LIN {X 0,Y 499.912,Z 1008.402,A -85,B 0,C 180,E1 21822.944,E2 21822.944} C_VEL
LIN {X 0,Y 504.848,Z 990.59,A -85,B 0,C 180,E1 21821.614,E2 21821.614} C_VEL
LIN {X 0,Y 509.783,Z 971.635,A -85,B 0,C 180,E1 21820.361,E2 21820.361} C_VEL
LIN {X 0,Y 514.878,Z 950.68,A -85,B 0,C 180,E1 21819.156,E2 21819.156} C_VEL
LIN {X 0,Y 520.634,Z 924.438,A -85,B 0,C 180,E1 21817.879,E2 21817.879} C_VEL
LIN {X 0,Y 525.094,Z 900.885,A -85,B 0,C 180,E1 21816.94,E2 21816.94} C_VEL
LIN {X 0,Y 528.641,Z 879.529,A -85,B 0,C 180,E1 21816.234,E2 21816.234} C_VEL
LIN {X 0,Y 531.615,Z 858.391,A -85,B 0,C 180,E1 21815.659,E2 21815.659} C_VEL
LIN {X 0,Y 534.308,Z 834.905,A -85,B 0,C 180,E1 21815.156,E2 21815.156} C_VEL
LIN {X 0,Y 536.742,Z 798.959,A -85,B 0,C 180,E1 21814.559,E2 21814.559} C_VEL
LIN {X 0,Y 548.311,Z 577.211,A -85,B 0,C 180,E1 21811.168,E2 21811.168} C_VEL
LIN {X 0,Y 553.738,Z 476.421,A -85,B 0,C 180,E1 21809.595,E2 21809.595} C_VEL
LIN {X 0,Y 544.019,Z 460.747,A -85,B 0,C 180,E1 21807.325,E2 21807.325} C_VEL
LIN {X 0,Y 534.97,Z 447.007,A -85,B 0,C 180,E1 21804.987,E2 21804.987} C_VEL
LIN {X 0,Y 526.575,Z 434.757,A -85,B 0,C 180,E1 21802.555,E2 21802.555} C_VEL
LIN {X 0,Y 521.092,Z 427.175,A -85,B 0,C 180,E1 21800.793,E2 21800.793} C_VEL
LIN {X 0,Y 517.186,Z 421.826,A -85,B 0,C 180,E1 21799.423,E2 21799.423} C_VEL
LIN {X 0,Y 512.336,Z 415.199,A -85,B 0,C 180,E1 21797.549,E2 21797.549} C_VEL
LIN {X 0,Y 507.667,Z 409.451,A -85,B 0,C 180,E1 21795.537,E2 21795.537} C_VEL
LIN {X 0,Y 506.729,Z 408.307,A -85,B 0,C 180,E1 21795.098,E2 21795.098} C_VEL
LIN {X 0,Y 503.193,Z 404.431,A -85,B 0,C 180,E1 21793.327,E2 21793.327} C_VEL
LIN {X 0,Y 502.048,Z 402.516,A -85,B 0,C 180,E1 21792.655,E2 21792.655} C_VEL
LIN {X 0,Y 498.77,Z 399.704,A -85,B 0,C 180,E1 21790.687,E2 21790.687} C_VEL
LIN {X 0,Y 496.811,Z 396.193,A -85,B 0,C 180,E1 21789.149,E2 21789.149} C_VEL
LIN {X 0,Y 493.046,Z 393.345,A -85,B 0,C 180,E1 21785.586,E2 21785.586} C_VEL
LIN {X 0,Y 491.629,Z 389.721,A -85,B 0,C 180,E1 21782.798,E2 21782.798} C_VEL
LIN {X 0,Y 491.752,Z 389.93,A -85,B 0,C 180,E1 21776.386,E2 21776.386} C_VEL
LIN {X 0,Y 492.937,Z 393.135,A -85,B 0,C 180,E1 21774.062,E2 21774.062} C_VEL
LIN {X 0,Y 496.449,Z 396.076,A -85,B 0,C 180,E1 21770.611,E2 21770.611} C_VEL
LIN {X 0,Y 497.033,Z 396.632,A -85,B 0,C 180,E1 21770.154,E2 21770.154} C_VEL
LIN {X 0,Y 499.129,Z 400.183,A -85,B 0,C 180,E1 21768.561,E2 21768.561} C_VEL
LIN {X 0,Y 502.365,Z 403.011,A -85,B 0,C 180,E1 21766.651,E2 21766.651} C_VEL
LIN {X 0,Y 505.237,Z 407.088,A -85,B 0,C 180,E1 21765.091,E2 21765.091} C_VEL
LIN {X 0,Y 507.467,Z 409.19,A -85,B 0,C 180,E1 21764.049,E2 21764.049} C_VEL
LIN {X 0,Y 510.926,Z 413.582,A -85,B 0,C 180,E1 21762.518,E2 21762.518} C_VEL
LIN {X 0,Y 512.597,Z 415.426,A -85,B 0,C 180,E1 21761.843,E2 21761.843} C_VEL
LIN {X 0,Y 517.532,Z 421.592,A -85,B 0,C 180,E1 21759.973,E2 21759.973} C_VEL
LIN {X 0,Y 522.294,Z 427.58,A -85,B 0,C 180,E1 21758.346,E2 21758.346} C_VEL
LIN {X 0,Y 526.558,Z 433.053,A -85,B 0,C 180,E1 21757.002,E2 21757.002} C_VEL
LIN {X 0,Y 534.048,Z 442.795,A -85,B 0,C 180,E1 21754.849,E2 21754.849} C_VEL
LIN {X 0,Y 542.616,Z 454.591,A -85,B 0,C 180,E1 21752.628,E2 21752.628} C_VEL
LIN {X 0,Y 551.517,Z 467.214,A -85,B 0,C 180,E1 21750.543,E2 21750.543} C_VEL
LIN {X 0,Y 553.74,Z 470.858,A -85,B 0,C 180,E1 21750.04,E2 21750.04} C_VEL
LIN {X 0,Y 542.052,Z 685.81,A -85,B 0,C 180,E1 21746.741,E2 21746.741} C_VEL
LIN {X 0,Y 535.822,Z 802.377,A -85,B 0,C 180,E1 21744.945,E2 21744.945} C_VEL
LIN {X 0,Y 533.339,Z 829.272,A -85,B 0,C 180,E1 21744.423,E2 21744.423} C_VEL
LIN {X 0,Y 529.817,Z 855.856,A -85,B 0,C 180,E1 21743.712,E2 21743.712} C_VEL
LIN {X 0,Y 526.549,Z 876.447,A -85,B 0,C 180,E1 21743.03,E2 21743.03} C_VEL
LIN {X 0,Y 522.905,Z 896.374,A -85,B 0,C 180,E1 21742.247,E2 21742.247} C_VEL
LIN {X 0,Y 518.74,Z 916.594,A -85,B 0,C 180,E1 21741.318,E2 21741.318} C_VEL
LIN {X 0,Y 514.01,Z 937.364,A -85,B 0,C 180,E1 21740.207,E2 21740.207} C_VEL
LIN {X 0,Y 507.632,Z 962.474,A -85,B 0,C 180,E1 21738.628,E2 21738.628} C_VEL
LIN {X 0,Y 501.992,Z 982.688,A -85,B 0,C 180,E1 21737.136,E2 21737.136} C_VEL
LIN {X 0,Y 496.85,Z 1000.115,A -85,B 0,C 180,E1 21735.676,E2 21735.676} C_VEL
LIN {X 0,Y 491.606,Z 1017.106,A -85,B 0,C 180,E1 21734.073,E2 21734.073} C_VEL
LIN {X 0,Y 486.038,Z 1034.545,A -85,B 0,C 180,E1 21732.217,E2 21732.217} C_VEL
LIN {X 0,Y 479.163,Z 1055.51,A -85,B 0,C 180,E1 21729.645,E2 21729.645} C_VEL
LIN {X 0,Y 473.899,Z 1071.228,A -85,B 0,C 180,E1 21727.419,E2 21727.419} C_VEL
LIN {X 0,Y 469.143,Z 1085.554,A -85,B 0,C 180,E1 21725.13,E2 21725.13} C_VEL
LIN {X 0,Y 464.525,Z 1099.816,A -85,B 0,C 180,E1 21722.555,E2 21722.555} C_VEL
LIN {X 0,Y 459.689,Z 1115.448,A -85,B 0,C 180,E1 21719.28,E2 21719.28} C_VEL
LIN {X 0,Y 459.025,Z 1117.597,A -85,B 0,C 180,E1 21718.78,E2 21718.78} C_VEL
LIN {X 0,Y 457.031,Z 1121.397,A -85,B 0,C 180,E1 21717.965,E2 21717.965} C_VEL
LIN {X 0,Y 448.52,Z 1131.236,A -85,B 0,C 180,E1 21715.841,E2 21715.841} C_VEL
LIN {X 0,Y 447.037,Z 1133.995,A -85,B 0,C 180,E1 21715.09,E2 21715.09} C_VEL
LIN {X 0,Y 444.634,Z 1143.256,A -85,B 0,C 180,E1 21712.196,E2 21712.196} C_VEL
LIN {X 0,Y 442.943,Z 1150.695,A -85,B 0,C 180,E1 21709.517,E2 21709.517} C_VEL
LIN {X 0,Y 441.679,Z 1157.301,A -85,B 0,C 180,E1 21706.742,E2 21706.742} C_VEL
LIN {X 0,Y 440.829,Z 1163.009,A -85,B 0,C 180,E1 21703.881,E2 21703.881} C_VEL
LIN {X 0,Y 440.237,Z 1168.647,A -85,B 0,C 180,E1 21700.336,E2 21700.336} C_VEL
LIN {X 0,Y 439.997,Z 1172.254,A -85,B 0,C 180,E1 21697.049,E2 21697.049} C_VEL
LIN {X 0,Y 439.929,Z 1174.329,A -85,B 0,C 180,E1 21694.171,E2 21694.171} C_VEL
LIN {X 0,Y 439.916,Z 1175.306,A -85,B 0,C 180,E1 21691.563,E2 21691.563} C_VEL
LIN {X 0,Y 439.916,Z 1175.409,A -85,B 0,C 180,E1 21688.958,E2 21688.958} C_VEL
LIN {X 0,Y 439.928,Z 1174.573,A -85,B 0,C 180,E1 21686.221,E2 21686.221} C_VEL
LIN {X 0,Y 439.98,Z 1172.771,A -85,B 0,C 180,E1 21683.476,E2 21683.476} C_VEL
LIN {X 0,Y 440.122,Z 1169.989,A -85,B 0,C 180,E1 21680.718,E2 21680.718} C_VEL
LIN {X 0,Y 440.447,Z 1166.205,A -85,B 0,C 180,E1 21677.945,E2 21677.945} C_VEL
LIN {X 0,Y 441.103,Z 1160.992,A -85,B 0,C 180,E1 21674.942,E2 21674.942} C_VEL
LIN {X 0,Y 442.567,Z 1152.645,A -85,B 0,C 180,E1 21671.151,E2 21671.151} C_VEL
LIN {X 0,Y 444.295,Z 1144.699,A -85,B 0,C 180,E1 21668.203,E2 21668.203} C_VEL
LIN {X 0,Y 446.381,Z 1136.332,A -85,B 0,C 180,E1 21665.519,E2 21665.519} C_VEL
LIN {X 0,Y 449.046,Z 1126.79,A -85,B 0,C 180,E1 21662.841,E2 21662.841} C_VEL
LIN {X 0,Y 452.729,Z 1114.867,A -85,B 0,C 180,E1 21659.912,E2 21659.912} C_VEL
LIN {X 0,Y 457.6,Z 1099.827,A -85,B 0,C 180,E1 21656.74,E2 21656.74} C_VEL
LIN {X 0,Y 462.204,Z 1086.291,A -85,B 0,C 180,E1 21654.263,E2 21654.263} C_VEL
LIN {X 0,Y 466.858,Z 1072.835,A -85,B 0,C 180,E1 21652.073,E2 21652.073} C_VEL
LIN {X 0,Y 472.19,Z 1057.515,A -85,B 0,C 180,E1 21649.858,E2 21649.858} C_VEL
LIN {X 0,Y 478.997,Z 1037.801,A -85,B 0,C 180,E1 21647.362,E2 21647.362} C_VEL
LIN {X 0,Y 485.502,Z 1018.081,A -85,B 0,C 180,E1 21645.225,E2 21645.225} C_VEL
LIN {X 0,Y 490.925,Z 1001.155,A -85,B 0,C 180,E1 21643.611,E2 21643.611} C_VEL
LIN {X 0,Y 496.235,Z 983.798,A -85,B 0,C 180,E1 21642.143,E2 21642.143} C_VEL
LIN {X 0,Y 501.578,Z 965.263,A -85,B 0,C 180,E1 21640.756,E2 21640.756} C_VEL
LIN {X 0,Y 508.144,Z 940.734,A -85,B 0,C 180,E1 21639.172,E2 21639.172} C_VEL
LIN {X 0,Y 513.483,Z 918.099,A -85,B 0,C 180,E1 21637.944,E2 21637.944} C_VEL
LIN {X 0,Y 517.761,Z 898.046,A -85,B 0,C 180,E1 21637.012,E2 21637.012} C_VEL
LIN {X 0,Y 521.64,Z 877.583,A -85,B 0,C 180,E1 21636.201,E2 21636.201} C_VEL
LIN {X 0,Y 525.123,Z 856.307,A -85,B 0,C 180,E1 21635.492,E2 21635.492} C_VEL
LIN {X 0,Y 528.747,Z 829.724,A -85,B 0,C 180,E1 21634.781,E2 21634.781} C_VEL
LIN {X 0,Y 531.309,Z 802.773,A -85,B 0,C 180,E1 21634.256,E2 21634.256} C_VEL
LIN {X 0,Y 537.398,Z 692.803,A -85,B 0,C 180,E1 21632.554,E2 21632.554} C_VEL
LIN {X 0,Y 549.515,Z 477.081,A -85,B 0,C 180,E1 21629.234,E2 21629.234} C_VEL
LIN {X 0,Y 549.54,Z 475.04,A -85,B 0,C 180,E1 21629.185,E2 21629.185} C_VEL
LIN {X 0,Y 540.335,Z 461.8,A -85,B 0,C 180,E1 21626.99,E2 21626.99} C_VEL
LIN {X 0,Y 531.088,Z 448.868,A -85,B 0,C 180,E1 21624.528,E2 21624.528} C_VEL
LIN {X 0,Y 522.239,Z 437.289,A -85,B 0,C 180,E1 21621.863,E2 21621.863} C_VEL
LIN {X 0,Y 518.024,Z 431.951,A -85,B 0,C 180,E1 21620.449,E2 21620.449} C_VEL
LIN {X 0,Y 513.95,Z 426.774,A -85,B 0,C 180,E1 21618.96,E2 21618.96} C_VEL
LIN {X 0,Y 509.921,Z 421.7,A -85,B 0,C 180,E1 21617.341,E2 21617.341} C_VEL
LIN {X 0,Y 506.344,Z 417.431,A -85,B 0,C 180,E1 21615.755,E2 21615.755} C_VEL
LIN {X 0,Y 505.081,Z 415.892,A -85,B 0,C 180,E1 21615.148,E2 21615.148} C_VEL
LIN {X 0,Y 501.861,Z 412.22,A -85,B 0,C 180,E1 21613.48,E2 21613.48} C_VEL
LIN {X 0,Y 500.543,Z 410.201,A -85,B 0,C 180,E1 21612.694,E2 21612.694} C_VEL
LIN {X 0,Y 497.092,Z 406.889,A -85,B 0,C 180,E1 21610.489,E2 21610.489} C_VEL
LIN {X 0,Y 495.664,Z 404.104,A -85,B 0,C 180,E1 21609.287,E2 21609.287} C_VEL
LIN {X 0,Y 491.91,Z 401.065,A -85,B 0,C 180,E1 21605.482,E2 21605.482} C_VEL
LIN {X 0,Y 490.704,Z 397.658,A -85,B 0,C 180,E1 21602.686,E2 21602.686} C_VEL
LIN {X 0,Y 490.802,Z 397.82,A -85,B 0,C 180,E1 21597.431,E2 21597.431} C_VEL
LIN {X 0,Y 492.462,Z 401.837,A -85,B 0,C 180,E1 21594.173,E2 21594.173} C_VEL
LIN {X 0,Y 495.879,Z 404.384,A -85,B 0,C 180,E1 21590.951,E2 21590.951} C_VEL
LIN {X 0,Y 498.399,Z 408.5,A -85,B 0,C 180,E1 21589.013,E2 21589.013} C_VEL
LIN {X 0,Y 501.04,Z 410.717,A -85,B 0,C 180,E1 21587.436,E2 21587.436} C_VEL
LIN {X 0,Y 504.069,Z 414.911,A -85,B 0,C 180,E1 21585.761,E2 21585.761} C_VEL
LIN {X 0,Y 506.142,Z 417.001,A -85,B 0,C 180,E1 21584.767,E2 21584.767} C_VEL
LIN {X 0,Y 509.665,Z 421.495,A -85,B 0,C 180,E1 21583.179,E2 21583.179} C_VEL
LIN {X 0,Y 514.337,Z 427.727,A -85,B 0,C 180,E1 21581.291,E2 21581.291} C_VEL
LIN {X 0,Y 518.996,Z 434.232,A -85,B 0,C 180,E1 21579.591,E2 21579.591} C_VEL
LIN {X 0,Y 524.613,Z 442.115,A -85,B 0,C 180,E1 21577.74,E2 21577.74} C_VEL
LIN {X 0,Y 533.804,Z 455.667,A -85,B 0,C 180,E1 21575.04,E2 21575.04} C_VEL
LIN {X 0,Y 542.974,Z 470.067,A -85,B 0,C 180,E1 21572.648,E2 21572.648} C_VEL
LIN {X 0,Y 549.68,Z 481.2,A -85,B 0,C 180,E1 21571.044,E2 21571.044} C_VEL
LIN {X 0,Y 537.951,Z 691.52,A -85,B 0,C 180,E1 21567.801,E2 21567.801} C_VEL
LIN {X 0,Y 530.83,Z 822.089,A -85,B 0,C 180,E1 21565.783,E2 21565.783} C_VEL
LIN {X 0,Y 528.193,Z 849.404,A -85,B 0,C 180,E1 21565.265,E2 21565.265} C_VEL
LIN {X 0,Y 524.46,Z 875.969,A -85,B 0,C 180,E1 21564.582,E2 21564.582} C_VEL
LIN {X 0,Y 520.839,Z 897.573,A -85,B 0,C 180,E1 21563.888,E2 21563.888} C_VEL
LIN {X 0,Y 516.962,Z 917.84,A -85,B 0,C 180,E1 21563.106,E2 21563.106} C_VEL
LIN {X 0,Y 512.59,Z 938.224,A -85,B 0,C 180,E1 21562.185,E2 21562.185} C_VEL
LIN {X 0,Y 506.938,Z 962.266,A -85,B 0,C 180,E1 21560.906,E2 21560.906} C_VEL
LIN {X 0,Y 500.544,Z 986.296,A -85,B 0,C 180,E1 21559.382,E2 21559.382} C_VEL
LIN {X 0,Y 495.148,Z 1005.224,A -85,B 0,C 180,E1 21557.997,E2 21557.997} C_VEL
LIN {X 0,Y 489.611,Z 1023.657,A -85,B 0,C 180,E1 21556.466,E2 21556.466} C_VEL
LIN {X 0,Y 483.812,Z 1042.239,A -85,B 0,C 180,E1 21554.715,E2 21554.715} C_VEL
LIN {X 0,Y 476.711,Z 1064.314,A -85,B 0,C 180,E1 21552.32,E2 21552.32} C_VEL
LIN {X 0,Y 471.001,Z 1081.529,A -85,B 0,C 180,E1 21550.16,E2 21550.16} C_VEL
LIN {X 0,Y 465.97,Z 1096.733,A -85,B 0,C 180,E1 21548.012,E2 21548.012} C_VEL
LIN {X 0,Y 461.4,Z 1110.664,A -85,B 0,C 180,E1 21545.809,E2 21545.809} C_VEL
LIN {X 0,Y 456.812,Z 1124.995,A -85,B 0,C 180,E1 21543.265,E2 21543.265} C_VEL
LIN {X 0,Y 451.799,Z 1141.559,A -85,B 0,C 180,E1 21539.864,E2 21539.864} C_VEL
LIN {X 0,Y 448.598,Z 1152.843,A -85,B 0,C 180,E1 21537.188,E2 21537.188} C_VEL
LIN {X 0,Y 446.003,Z 1162.97,A -85,B 0,C 180,E1 21534.465,E2 21534.465} C_VEL
LIN {X 0,Y 444.025,Z 1171.642,A -85,B 0,C 180,E1 21531.811,E2 21531.811} C_VEL
LIN {X 0,Y 442.381,Z 1180.02,A -85,B 0,C 180,E1 21528.857,E2 21528.857} C_VEL
LIN {X 0,Y 441.026,Z 1188.768,A -85,B 0,C 180,E1 21525.113,E2 21525.113} C_VEL
LIN {X 0,Y 440.386,Z 1194.411,A -85,B 0,C 180,E1 21522.057,E2 21522.057} C_VEL
LIN {X 0,Y 440.099,Z 1198.284,A -85,B 0,C 180,E1 21519.414,E2 21519.414} C_VEL
LIN {X 0,Y 439.966,Z 1201.265,A -85,B 0,C 180,E1 21516.707,E2 21516.707} C_VEL
LIN {X 0,Y 439.922,Z 1203.156,A -85,B 0,C 180,E1 21514.171,E2 21514.171} C_VEL
LIN {X 0,Y 439.919,Z 1204.182,A -85,B 0,C 180,E1 21511.563,E2 21511.563} C_VEL
LIN {X 0,Y 439.918,Z 1204.275,A -85,B 0,C 180,E1 21508.958,E2 21508.958} C_VEL
LIN {X 0,Y 439.921,Z 1203.436,A -85,B 0,C 180,E1 21506.351,E2 21506.351} C_VEL
LIN {X 0,Y 439.956,Z 1201.661,A -85,B 0,C 180,E1 21503.737,E2 21503.737} C_VEL
LIN {X 0,Y 440.064,Z 1198.942,A -85,B 0,C 180,E1 21501.112,E2 21501.112} C_VEL
LIN {X 0,Y 440.302,Z 1195.262,A -85,B 0,C 180,E1 21498.473,E2 21498.473} C_VEL
LIN {X 0,Y 440.826,Z 1190.339,A -85,B 0,C 180,E1 21495.687,E2 21495.687} C_VEL
LIN {X 0,Y 441.601,Z 1184.614,A -85,B 0,C 180,E1 21493.018,E2 21493.018} C_VEL
LIN {X 0,Y 442.848,Z 1177.481,A -85,B 0,C 180,E1 21490.204,E2 21490.204} C_VEL
LIN {X 0,Y 444.98,Z 1167.492,A -85,B 0,C 180,E1 21486.845,E2 21486.845} C_VEL
LIN {X 0,Y 447.908,Z 1155.482,A -85,B 0,C 180,E1 21483.484,E2 21483.484} C_VEL
LIN {X 0,Y 450.918,Z 1144.49,A -85,B 0,C 180,E1 21480.802,E2 21480.802} C_VEL
LIN {X 0,Y 454.409,Z 1132.778,A -85,B 0,C 180,E1 21478.272,E2 21478.272} C_VEL
LIN {X 0,Y 458.714,Z 1118.999,A -85,B 0,C 180,E1 21475.63,E2 21475.63} C_VEL
LIN {X 0,Y 464.839,Z 1100.155,A -85,B 0,C 180,E1 21472.503,E2 21472.503} C_VEL
LIN {X 0,Y 469.959,Z 1084.615,A -85,B 0,C 180,E1 21470.259,E2 21470.259} C_VEL
LIN {X 0,Y 475.065,Z 1069.163,A -85,B 0,C 180,E1 21468.27,E2 21468.27} C_VEL
LIN {X 0,Y 480.327,Z 1053.064,A -85,B 0,C 180,E1 21466.422,E2 21466.422} C_VEL
LIN {X 0,Y 486.799,Z 1032.9,A -85,B 0,C 180,E1 21464.376,E2 21464.376} C_VEL
LIN {X 0,Y 493.628,Z 1010.39,A -85,B 0,C 180,E1 21462.417,E2 21462.417} C_VEL
LIN {X 0,Y 499.161,Z 991.133,A -85,B 0,C 180,E1 21460.961,E2 21460.961} C_VEL
LIN {X 0,Y 504.246,Z 972.268,A -85,B 0,C 180,E1 21459.704,E2 21459.704} C_VEL
LIN {X 0,Y 509.328,Z 952.048,A -85,B 0,C 180,E1 21458.529,E2 21458.529} C_VEL
LIN {X 0,Y 514.893,Z 927.87,A -85,B 0,C 180,E1 21457.326,E2 21457.326} C_VEL
LIN {X 0,Y 519.986,Z 902.097,A -85,B 0,C 180,E1 21456.278,E2 21456.278} C_VEL
LIN {X 0,Y 523.759,Z 880.125,A -85,B 0,C 180,E1 21455.546,E2 21455.546} C_VEL
LIN {X 0,Y 526.846,Z 858.886,A -85,B 0,C 180,E1 21454.965,E2 21454.965} C_VEL
LIN {X 0,Y 529.517,Z 836.418,A -85,B 0,C 180,E1 21454.479,E2 21454.479} C_VEL
LIN {X 0,Y 531.799,Z 806.687,A -85,B 0,C 180,E1 21453.968,E2 21453.968} C_VEL
LIN {X 0,Y 543.813,Z 583.563,A -85,B 0,C 180,E1 21450.544,E2 21450.544} C_VEL
LIN {X 0,Y 549.559,Z 480.937,A -85,B 0,C 180,E1 21448.945,E2 21448.945} C_VEL
LIN {X 0,Y 541.033,Z 467.045,A -85,B 0,C 180,E1 21446.893,E2 21446.893} C_VEL
LIN {X 0,Y 532.508,Z 453.893,A -85,B 0,C 180,E1 21444.636,E2 21444.636} C_VEL
LIN {X 0,Y 523.69,Z 440.758,A -85,B 0,C 180,E1 21442.006,E2 21442.006} C_VEL
LIN {X 0,Y 516.206,Z 430.294,A -85,B 0,C 180,E1 21439.461,E2 21439.461} C_VEL
LIN {X 0,Y 510.049,Z 421.85,A -85,B 0,C 180,E1 21437.042,E2 21437.042} C_VEL
LIN {X 0,Y 506.435,Z 417.562,A -85,B 0,C 180,E1 21435.459,E2 21435.459} C_VEL
LIN {X 0,Y 505.288,Z 416.012,A -85,B 0,C 180,E1 21434.907,E2 21434.907} C_VEL
LIN {X 0,Y 501.71,Z 411.973,A -85,B 0,C 180,E1 21433.074,E2 21433.074} C_VEL
LIN {X 0,Y 500.674,Z 410.284,A -85,B 0,C 180,E1 21432.456,E2 21432.456} C_VEL
LIN {X 0,Y 497.466,Z 407.395,A -85,B 0,C 180,E1 21430.481,E2 21430.481} C_VEL
LIN {X 0,Y 495.538,Z 404.029,A -85,B 0,C 180,E1 21428.938,E2 21428.938} C_VEL
LIN {X 0,Y 491.819,Z 400.953,A -85,B 0,C 180,E1 21425.249,E2 21425.249} C_VEL
LIN {X 0,Y 490.604,Z 397.655,A -85,B 0,C 180,E1 21422.687,E2 21422.687} C_VEL
LIN {X 0,Y 490.727,Z 397.822,A -85,B 0,C 180,E1 21416.495,E2 21416.495} C_VEL
LIN {X 0,Y 491.877,Z 401.014,A -85,B 0,C 180,E1 21414.166,E2 21414.166} C_VEL
LIN {X 0,Y 495.336,Z 403.967,A -85,B 0,C 180,E1 21410.707,E2 21410.707} C_VEL
LIN {X 0,Y 495.897,Z 404.652,A -85,B 0,C 180,E1 21410.249,E2 21410.249} C_VEL
LIN {X 0,Y 498.157,Z 408.263,A -85,B 0,C 180,E1 21408.538,E2 21408.538} C_VEL
LIN {X 0,Y 500.991,Z 410.741,A -85,B 0,C 180,E1 21406.849,E2 21406.849} C_VEL
LIN {X 0,Y 503.933,Z 414.892,A -85,B 0,C 180,E1 21405.228,E2 21405.228} C_VEL
LIN {X 0,Y 506.021,Z 416.947,A -85,B 0,C 180,E1 21404.235,E2 21404.235} C_VEL
LIN {X 0,Y 509.568,Z 421.394,A -85,B 0,C 180,E1 21402.647,E2 21402.647} C_VEL
LIN {X 0,Y 511.144,Z 423.284,A -85,B 0,C 180,E1 21401.996,E2 21401.996} C_VEL
LIN {X 0,Y 515.816,Z 429.165,A -85,B 0,C 180,E1 21400.199,E2 21400.199} C_VEL
LIN {X 0,Y 520.521,Z 435.161,A -85,B 0,C 180,E1 21398.564,E2 21398.564} C_VEL
LIN {X 0,Y 524.736,Z 440.655,A -85,B 0,C 180,E1 21397.214,E2 21397.214} C_VEL
LIN {X 0,Y 532.057,Z 450.329,A -85,B 0,C 180,E1 21395.075,E2 21395.075} C_VEL
LIN {X 0,Y 541.933,Z 464.002,A -85,B 0,C 180,E1 21392.502,E2 21392.502} C_VEL
LIN {X 0,Y 549.547,Z 475.251,A -85,B 0,C 180,E1 21390.7,E2 21390.7} C_VEL
LIN {X 0,Y 537.465,Z 690.469,A -85,B 0,C 180,E1 21387.387,E2 21387.387} C_VEL
LIN {X 0,Y 531.264,Z 802.665,A -85,B 0,C 180,E1 21385.652,E2 21385.652} C_VEL
LIN {X 0,Y 528.699,Z 829.702,A -85,B 0,C 180,E1 21385.126,E2 21385.126} C_VEL
LIN {X 0,Y 525.085,Z 856.24,A -85,B 0,C 180,E1 21384.416,E2 21384.416} C_VEL
LIN {X 0,Y 521.745,Z 876.722,A -85,B 0,C 180,E1 21383.737,E2 21383.737} C_VEL
LIN {X 0,Y 518,Z 896.649,A -85,B 0,C 180,E1 21382.954,E2 21382.954} C_VEL
LIN {X 0,Y 513.715,Z 916.867,A -85,B 0,C 180,E1 21382.023,E2 21382.023} C_VEL
LIN {X 0,Y 508.732,Z 938.119,A -85,B 0,C 180,E1 21380.882,E2 21380.882} C_VEL
LIN {X 0,Y 502.041,Z 963.551,A -85,B 0,C 180,E1 21379.27,E2 21379.27} C_VEL
LIN {X 0,Y 496.455,Z 982.963,A -85,B 0,C 180,E1 21377.829,E2 21377.829} C_VEL
LIN {X 0,Y 491.098,Z 1000.508,A -85,B 0,C 180,E1 21376.353,E2 21376.353} C_VEL
LIN {X 0,Y 485.677,Z 1017.467,A -85,B 0,C 180,E1 21374.743,E2 21374.743} C_VEL
LIN {X 0,Y 479.695,Z 1035.544,A -85,B 0,C 180,E1 21372.801,E2 21372.801} C_VEL
LIN {X 0,Y 472.544,Z 1056.483,A -85,B 0,C 180,E1 21370.192,E2 21370.192} C_VEL
LIN {X 0,Y 467.315,Z 1071.504,A -85,B 0,C 180,E1 21368.039,E2 21368.039} C_VEL
LIN {X 0,Y 462.621,Z 1085.073,A -85,B 0,C 180,E1 21365.853,E2 21365.853} C_VEL
LIN {X 0,Y 458.201,Z 1098.029,A -85,B 0,C 180,E1 21363.51,E2 21363.51} C_VEL
LIN {X 0,Y 453.76,Z 1111.547,A -85,B 0,C 180,E1 21360.744,E2 21360.744} C_VEL
LIN {X 0,Y 449.448,Z 1125.473,A -85,B 0,C 180,E1 21357.419,E2 21357.419} C_VEL
LIN {X 0,Y 447.037,Z 1133.995,A -85,B 0,C 180,E1 21355.09,E2 21355.09} C_VEL
LIN {X 0,Y 445.245,Z 1137.162,A -85,B 0,C 180,E1 21354.208,E2 21354.208} C_VEL
LIN {X 0,Y 437.242,Z 1145.592,A -85,B 0,C 180,E1 21351.896,E2 21351.896} C_VEL
LIN {X 0,Y 435.932,Z 1147.901,A -85,B 0,C 180,E1 21351.092,E2 21351.092} C_VEL
LIN {X 0,Y 434.05,Z 1156.467,A -85,B 0,C 180,E1 21347.564,E2 21347.564} C_VEL
LIN {X 0,Y 433.058,Z 1162.235,A -85,B 0,C 180,E1 21344.713,E2 21344.713} C_VEL
LIN {X 0,Y 432.444,Z 1166.938,A -85,B 0,C 180,E1 21341.875,E2 21341.875} C_VEL
LIN {X 0,Y 432.135,Z 1170.458,A -85,B 0,C 180,E1 21339.187,E2 21339.187} C_VEL
LIN {X 0,Y 431.99,Z 1173.068,A -85,B 0,C 180,E1 21336.512,E2 21336.512} C_VEL
LIN {X 0,Y 431.933,Z 1174.79,A -85,B 0,C 180,E1 21333.849,E2 21333.849} C_VEL
LIN {X 0,Y 431.922,Z 1175.634,A -85,B 0,C 180,E1 21331.194,E2 21331.194} C_VEL
LIN {X 0,Y 431.921,Z 1175.606,A -85,B 0,C 180,E1 21328.541,E2 21328.541} C_VEL
LIN {X 0,Y 431.936,Z 1174.704,A -85,B 0,C 180,E1 21325.885,E2 21325.885} C_VEL
LIN {X 0,Y 431.992,Z 1172.909,A -85,B 0,C 180,E1 21323.202,E2 21323.202} C_VEL
LIN {X 0,Y 432.161,Z 1170.099,A -85,B 0,C 180,E1 21320.411,E2 21320.411} C_VEL
LIN {X 0,Y 432.547,Z 1166.071,A -85,B 0,C 180,E1 21317.45,E2 21317.45} C_VEL
LIN {X 0,Y 433.503,Z 1159.61,A -85,B 0,C 180,E1 21313.795,E2 21313.795} C_VEL
LIN {X 0,Y 434.986,Z 1151.881,A -85,B 0,C 180,E1 21310.391,E2 21310.391} C_VEL
LIN {X 0,Y 436.807,Z 1144.178,A -85,B 0,C 180,E1 21307.526,E2 21307.526} C_VEL
LIN {X 0,Y 439.228,Z 1135.244,A -85,B 0,C 180,E1 21304.657,E2 21304.657} C_VEL
LIN {X 0,Y 442.983,Z 1122.999,A -85,B 0,C 180,E1 21301.265,E2 21301.265} C_VEL
LIN {X 0,Y 447.339,Z 1109.627,A -85,B 0,C 180,E1 21298.144,E2 21298.144} C_VEL
LIN {X 0,Y 451.619,Z 1097.346,A -85,B 0,C 180,E1 21295.629,E2 21295.629} C_VEL
LIN {X 0,Y 456.281,Z 1084.29,A -85,B 0,C 180,E1 21293.257,E2 21293.257} C_VEL
LIN {X 0,Y 462.532,Z 1067.138,A -85,B 0,C 180,E1 21290.512,E2 21290.512} C_VEL
LIN {X 0,Y 469.273,Z 1048.173,A -85,B 0,C 180,E1 21287.926,E2 21287.926} C_VEL
LIN {X 0,Y 474.953,Z 1032.044,A -85,B 0,C 180,E1 21285.996,E2 21285.996} C_VEL
LIN {X 0,Y 480.673,Z 1015.343,A -85,B 0,C 180,E1 21284.226,E2 21284.226} C_VEL
LIN {X 0,Y 487.439,Z 994.816,A -85,B 0,C 180,E1 21282.313,E2 21282.313} C_VEL
LIN {X 0,Y 494.524,Z 971.532,A -85,B 0,C 180,E1 21280.469,E2 21280.469} C_VEL
LIN {X 0,Y 500.073,Z 951.864,A -85,B 0,C 180,E1 21279.125,E2 21279.125} C_VEL
LIN {X 0,Y 505.263,Z 932.019,A -85,B 0,C 180,E1 21277.947,E2 21277.947} C_VEL
LIN {X 0,Y 510.079,Z 911.622,A -85,B 0,C 180,E1 21276.893,E2 21276.893} C_VEL
LIN {X 0,Y 515.728,Z 884.461,A -85,B 0,C 180,E1 21275.724,E2 21275.724} C_VEL
LIN {X 0,Y 519.774,Z 861.161,A -85,B 0,C 180,E1 21274.914,E2 21274.914} C_VEL
LIN {X 0,Y 522.895,Z 839.751,A -85,B 0,C 180,E1 21274.305,E2 21274.305} C_VEL
LIN {X 0,Y 525.433,Z 818.339,A -85,B 0,C 180,E1 21273.819,E2 21273.819} C_VEL
LIN {X 0,Y 527.636,Z 792.245,A -85,B 0,C 180,E1 21273.356,E2 21273.356} C_VEL
LIN {X 0,Y 540.214,Z 569.172,A -85,B 0,C 180,E1 21269.921,E2 21269.921} C_VEL
LIN {X 0,Y 545.457,Z 479.792,A -85,B 0,C 180,E1 21268.53,E2 21268.53} C_VEL
LIN {X 0,Y 535.139,Z 464.787,A -85,B 0,C 180,E1 21265.957,E2 21265.957} C_VEL
LIN {X 0,Y 527.262,Z 454.048,A -85,B 0,C 180,E1 21263.765,E2 21263.765} C_VEL
LIN {X 0,Y 520.299,Z 444.653,A -85,B 0,C 180,E1 21261.594,E2 21261.594} C_VEL
LIN {X 0,Y 515.994,Z 439.147,A -85,B 0,C 180,E1 21260.118,E2 21260.118} C_VEL
LIN {X 0,Y 512.274,Z 434.32,A -85,B 0,C 180,E1 21258.728,E2 21258.728} C_VEL
LIN {X 0,Y 508.171,Z 429.155,A -85,B 0,C 180,E1 21257.048,E2 21257.048} C_VEL
LIN {X 0,Y 504.567,Z 424.613,A -85,B 0,C 180,E1 21255.399,E2 21255.399} C_VEL
LIN {X 0,Y 500.298,Z 419.609,A -85,B 0,C 180,E1 21253.17,E2 21253.17} C_VEL
LIN {X 0,Y 499.384,Z 418.079,A -85,B 0,C 180,E1 21252.606,E2 21252.606} C_VEL
LIN {X 0,Y 495.958,Z 414.809,A -85,B 0,C 180,E1 21250.395,E2 21250.395} C_VEL
LIN {X 0,Y 494.403,Z 411.931,A -85,B 0,C 180,E1 21249.076,E2 21249.076} C_VEL
LIN {X 0,Y 490.781,Z 408.828,A -85,B 0,C 180,E1 21245.26,E2 21245.26} C_VEL
LIN {X 0,Y 489.689,Z 405.594,A -85,B 0,C 180,E1 21242.575,E2 21242.575} C_VEL
LIN {X 0,Y 489.786,Z 405.716,A -85,B 0,C 180,E1 21237.543,E2 21237.543} C_VEL
LIN {X 0,Y 491.486,Z 409.825,A -85,B 0,C 180,E1 21234.162,E2 21234.162} C_VEL
LIN {X 0,Y 494.688,Z 412.23,A -85,B 0,C 180,E1 21231.105,E2 21231.105} C_VEL
LIN {X 0,Y 497.255,Z 416.391,A -85,B 0,C 180,E1 21229.105,E2 21229.105} C_VEL
LIN {X 0,Y 499.764,Z 418.606,A -85,B 0,C 180,E1 21227.58,E2 21227.58} C_VEL
LIN {X 0,Y 502.99,Z 422.931,A -85,B 0,C 180,E1 21225.788,E2 21225.788} C_VEL
LIN {X 0,Y 504.695,Z 424.739,A -85,B 0,C 180,E1 21224.957,E2 21224.957} C_VEL
LIN {X 0,Y 508.31,Z 429.304,A -85,B 0,C 180,E1 21223.31,E2 21223.31} C_VEL
LIN {X 0,Y 512.926,Z 435.691,A -85,B 0,C 180,E1 21221.414,E2 21221.414} C_VEL
LIN {X 0,Y 519.084,Z 444.288,A -85,B 0,C 180,E1 21219.182,E2 21219.182} C_VEL
LIN {X 0,Y 526.497,Z 455.289,A -85,B 0,C 180,E1 21216.802,E2 21216.802} C_VEL
LIN {X 0,Y 534.421,Z 467.383,A -85,B 0,C 180,E1 21214.541,E2 21214.541} C_VEL
LIN {X 0,Y 543.827,Z 482.605,A -85,B 0,C 180,E1 21212.13,E2 21212.13} C_VEL
LIN {X 0,Y 545.542,Z 485.664,A -85,B 0,C 180,E1 21211.711,E2 21211.711} C_VEL
LIN {X 0,Y 533.343,Z 697.786,A -85,B 0,C 180,E1 21208.432,E2 21208.432} C_VEL
LIN {X 0,Y 526.337,Z 821.952,A -85,B 0,C 180,E1 21206.506,E2 21206.506} C_VEL
LIN {X 0,Y 523.605,Z 849.464,A -85,B 0,C 180,E1 21205.983,E2 21205.983} C_VEL
LIN {X 0,Y 519.767,Z 875.982,A -85,B 0,C 180,E1 21205.301,E2 21205.301} C_VEL
LIN {X 0,Y 516.195,Z 896.802,A -85,B 0,C 180,E1 21204.633,E2 21204.633} C_VEL
LIN {X 0,Y 512.136,Z 917.451,A -85,B 0,C 180,E1 21203.841,E2 21203.841} C_VEL
LIN {X 0,Y 507.616,Z 937.962,A -85,B 0,C 180,E1 21202.914,E2 21202.914} C_VEL
LIN {X 0,Y 501.789,Z 962.001,A -85,B 0,C 180,E1 21201.636,E2 21201.636} C_VEL
LIN {X 0,Y 495.192,Z 986.028,A -85,B 0,C 180,E1 21200.109,E2 21200.109} C_VEL
LIN {X 0,Y 489.62,Z 1004.955,A -85,B 0,C 180,E1 21198.72,E2 21198.72} C_VEL
LIN {X 0,Y 483.83,Z 1023.606,A -85,B 0,C 180,E1 21197.163,E2 21197.163} C_VEL
LIN {X 0,Y 477.714,Z 1042.521,A -85,B 0,C 180,E1 21195.367,E2 21195.367} C_VEL
LIN {X 0,Y 469.977,Z 1065.582,A -85,B 0,C 180,E1 21192.822,E2 21192.822} C_VEL
LIN {X 0,Y 464.243,Z 1082.224,A -85,B 0,C 180,E1 21190.699,E2 21190.699} C_VEL
LIN {X 0,Y 459.043,Z 1097.316,A -85,B 0,C 180,E1 21188.532,E2 21188.532} C_VEL
LIN {X 0,Y 454.044,Z 1111.956,A -85,B 0,C 180,E1 21186.169,E2 21186.169} C_VEL
LIN {X 0,Y 448.285,Z 1129.263,A -85,B 0,C 180,E1 21182.971,E2 21182.971} C_VEL
LIN {X 0,Y 444.131,Z 1142.453,A -85,B 0,C 180,E1 21180.134,E2 21180.134} C_VEL
LIN {X 0,Y 440.829,Z 1153.62,A -85,B 0,C 180,E1 21177.415,E2 21177.415} C_VEL
LIN {X 0,Y 438.182,Z 1163.51,A -85,B 0,C 180,E1 21174.682,E2 21174.682} C_VEL
LIN {X 0,Y 435.761,Z 1173.859,A -85,B 0,C 180,E1 21171.397,E2 21171.397} C_VEL
LIN {X 0,Y 433.931,Z 1183.098,A -85,B 0,C 180,E1 21167.846,E2 21167.846} C_VEL
LIN {X 0,Y 432.954,Z 1189.546,A -85,B 0,C 180,E1 21164.853,E2 21164.853} C_VEL
LIN {X 0,Y 432.398,Z 1194.357,A -85,B 0,C 180,E1 21162.147,E2 21162.147} C_VEL
LIN {X 0,Y 432.102,Z 1198.183,A -85,B 0,C 180,E1 21159.456,E2 21159.456} C_VEL
LIN {X 0,Y 431.968,Z 1201.054,A -85,B 0,C 180,E1 21156.771,E2 21156.771} C_VEL
LIN {X 0,Y 431.925,Z 1202.963,A -85,B 0,C 180,E1 21154.115,E2 21154.115} C_VEL
LIN {X 0,Y 431.923,Z 1203.943,A -85,B 0,C 180,E1 21151.459,E2 21151.459} C_VEL
LIN {X 0,Y 431.922,Z 1204.013,A -85,B 0,C 180,E1 21148.939,E2 21148.939} C_VEL
LIN {X 0,Y 431.923,Z 1203.173,A -85,B 0,C 180,E1 21146.284,E2 21146.284} C_VEL
LIN {X 0,Y 431.962,Z 1201.397,A -85,B 0,C 180,E1 21143.621,E2 21143.621} C_VEL
LIN {X 0,Y 432.074,Z 1198.676,A -85,B 0,C 180,E1 21140.946,E2 21140.946} C_VEL
LIN {X 0,Y 432.334,Z 1194.995,A -85,B 0,C 180,E1 21138.257,E2 21138.257} C_VEL
LIN {X 0,Y 432.855,Z 1190.331,A -85,B 0,C 180,E1 21135.554,E2 21135.554} C_VEL
LIN {X 0,Y 433.67,Z 1184.655,A -85,B 0,C 180,E1 21132.836,E2 21132.836} C_VEL
LIN {X 0,Y 434.969,Z 1177.572,A -85,B 0,C 180,E1 21129.971,E2 21129.971} C_VEL
LIN {X 0,Y 436.902,Z 1168.78,A -85,B 0,C 180,E1 21126.929,E2 21126.929} C_VEL
LIN {X 0,Y 440.254,Z 1155.731,A -85,B 0,C 180,E1 21123.131,E2 21123.131} C_VEL
LIN {X 0,Y 443.404,Z 1144.797,A -85,B 0,C 180,E1 21120.407,E2 21120.407} C_VEL
LIN {X 0,Y 447.036,Z 1133.147,A -85,B 0,C 180,E1 21117.838,E2 21117.838} C_VEL
LIN {X 0,Y 451.269,Z 1120.145,A -85,B 0,C 180,E1 21115.29,E2 21115.29} C_VEL
LIN {X 0,Y 457.055,Z 1103.21,A -85,B 0,C 180,E1 21112.368,E2 21112.368} C_VEL
LIN {X 0,Y 463.184,Z 1085.276,A -85,B 0,C 180,E1 21109.72,E2 21109.72} C_VEL
LIN {X 0,Y 468.48,Z 1069.87,A -85,B 0,C 180,E1 21107.707,E2 21107.707} C_VEL
LIN {X 0,Y 473.944,Z 1053.785,A -85,B 0,C 180,E1 21105.833,E2 21105.833} C_VEL
LIN {X 0,Y 479.737,Z 1036.316,A -85,B 0,C 180,E1 21104.025,E2 21104.025} C_VEL
LIN {X 0,Y 486.975,Z 1013.786,A -85,B 0,C 180,E1 21101.99,E2 21101.99} C_VEL
LIN {X 0,Y 493.541,Z 991.674,A -85,B 0,C 180,E1 21100.293,E2 21100.293} C_VEL
LIN {X 0,Y 498.776,Z 972.899,A -85,B 0,C 180,E1 21099.032,E2 21099.032} C_VEL
LIN {X 0,Y 503.746,Z 953.798,A -85,B 0,C 180,E1 21097.91,E2 21097.91} C_VEL
LIN {X 0,Y 508.388,Z 934.423,A -85,B 0,C 180,E1 21096.92,E2 21096.92} C_VEL
LIN {X 0,Y 512.905,Z 913.55,A -85,B 0,C 180,E1 21096.002,E2 21096.002} C_VEL
LIN {X 0,Y 518.02,Z 886.601,A -85,B 0,C 180,E1 21095.023,E2 21095.023} C_VEL
LIN {X 0,Y 521.878,Z 861.445,A -85,B 0,C 180,E1 21094.309,E2 21094.309} C_VEL
LIN {X 0,Y 524.633,Z 839.466,A -85,B 0,C 180,E1 21093.82,E2 21093.82} C_VEL
LIN {X 0,Y 526.66,Z 816.733,A -85,B 0,C 180,E1 21093.411,E2 21093.411} C_VEL
LIN {X 0,Y 538.89,Z 598.341,A -85,B 0,C 180,E1 21090.039,E2 21090.039} C_VEL
LIN {X 0,Y 545.459,Z 485.383,A -85,B 0,C 180,E1 21088.285,E2 21088.285} C_VEL
LIN {X 0,Y 537.031,Z 471.684,A -85,B 0,C 180,E1 21086.185,E2 21086.185} C_VEL
LIN {X 0,Y 529.71,Z 460.26,A -85,B 0,C 180,E1 21084.181,E2 21084.181} C_VEL
LIN {X 0,Y 521.559,Z 447.909,A -85,B 0,C 180,E1 21081.686,E2 21081.686} C_VEL
LIN {X 0,Y 514.202,Z 437.479,A -85,B 0,C 180,E1 21079.127,E2 21079.127} C_VEL
LIN {X 0,Y 508.421,Z 429.423,A -85,B 0,C 180,E1 21076.804,E2 21076.804} C_VEL
LIN {X 0,Y 504.759,Z 424.925,A -85,B 0,C 180,E1 21075.158,E2 21075.158} C_VEL
LIN {X 0,Y 503.62,Z 423.525,A -85,B 0,C 180,E1 21074.605,E2 21074.605} C_VEL
LIN {X 0,Y 500.143,Z 419.359,A -85,B 0,C 180,E1 21072.763,E2 21072.763} C_VEL
LIN {X 0,Y 499.271,Z 418.025,A -85,B 0,C 180,E1 21072.236,E2 21072.236} C_VEL
LIN {X 0,Y 496.091,Z 414.971,A -85,B 0,C 180,E1 21070.217,E2 21070.217} C_VEL
LIN {X 0,Y 494.422,Z 411.923,A -85,B 0,C 180,E1 21068.841,E2 21068.841} C_VEL
LIN {X 0,Y 490.761,Z 408.831,A -85,B 0,C 180,E1 21065.143,E2 21065.143} C_VEL
LIN {X 0,Y 489.58,Z 405.589,A -85,B 0,C 180,E1 21062.575,E2 21062.575} C_VEL
LIN {X 0,Y 489.704,Z 405.716,A -85,B 0,C 180,E1 21056.605,E2 21056.605} C_VEL
LIN {X 0,Y 490.818,Z 408.893,A -85,B 0,C 180,E1 21054.271,E2 21054.271} C_VEL
LIN {X 0,Y 494.223,Z 411.857,A -85,B 0,C 180,E1 21050.803,E2 21050.803} C_VEL
LIN {X 0,Y 494.829,Z 412.798,A -85,B 0,C 180,E1 21050.286,E2 21050.286} C_VEL
LIN {X 0,Y 497.186,Z 416.33,A -85,B 0,C 180,E1 21048.516,E2 21048.516} C_VEL
LIN {X 0,Y 499.714,Z 418.64,A -85,B 0,C 180,E1 21046.991,E2 21046.991} C_VEL
LIN {X 0,Y 502.855,Z 422.914,A -85,B 0,C 180,E1 21045.255,E2 21045.255} C_VEL
LIN {X 0,Y 504.574,Z 424.686,A -85,B 0,C 180,E1 21044.424,E2 21044.424} C_VEL
LIN {X 0,Y 508.345,Z 429.324,A -85,B 0,C 180,E1 21042.722,E2 21042.722} C_VEL
LIN {X 0,Y 514.039,Z 436.631,A -85,B 0,C 180,E1 21040.454,E2 21040.454} C_VEL
LIN {X 0,Y 518.833,Z 442.842,A -85,B 0,C 180,E1 21038.758,E2 21038.758} C_VEL
LIN {X 0,Y 525.11,Z 451.03,A -85,B 0,C 180,E1 21036.757,E2 21036.757} C_VEL
LIN {X 0,Y 534.009,Z 463.321,A -85,B 0,C 180,E1 21034.223,E2 21034.223} C_VEL
LIN {X 0,Y 542.617,Z 475.745,A -85,B 0,C 180,E1 21032.032,E2 21032.032} C_VEL
LIN {X 0,Y 545.4,Z 480.1,A -85,B 0,C 180,E1 21031.362,E2 21031.362} C_VEL
LIN {X 0,Y 532.935,Z 695.343,A -85,B 0,C 180,E1 21028.042,E2 21028.042} C_VEL
LIN {X 0,Y 526.781,Z 803.059,A -85,B 0,C 180,E1 21026.369,E2 21026.369} C_VEL
LIN {X 0,Y 524.123,Z 830.268,A -85,B 0,C 180,E1 21025.838,E2 21025.838} C_VEL
LIN {X 0,Y 520.434,Z 856.624,A -85,B 0,C 180,E1 21025.132,E2 21025.132} C_VEL
LIN {X 0,Y 516.888,Z 877.731,A -85,B 0,C 180,E1 21024.43,E2 21024.43} C_VEL
LIN {X 0,Y 512.914,Z 898.2,A -85,B 0,C 180,E1 21023.619,E2 21023.619} C_VEL
LIN {X 0,Y 508.266,Z 919.386,A -85,B 0,C 180,E1 21022.631,E2 21022.631} C_VEL
LIN {X 0,Y 501.78,Z 945.528,A -85,B 0,C 180,E1 21021.179,E2 21021.179} C_VEL
LIN {X 0,Y 496.036,Z 966.236,A -85,B 0,C 180,E1 21019.813,E2 21019.813} C_VEL
LIN {X 0,Y 490.539,Z 984.691,A -85,B 0,C 180,E1 21018.422,E2 21018.422} C_VEL
LIN {X 0,Y 485.089,Z 1001.92,A -85,B 0,C 180,E1 21016.953,E2 21016.953} C_VEL
LIN {X 0,Y 479.28,Z 1019.46,A -85,B 0,C 180,E1 21015.262,E2 21015.262} C_VEL
LIN {X 0,Y 472.208,Z 1040.096,A -85,B 0,C 180,E1 21012.985,E2 21012.985} C_VEL
LIN {X 0,Y 465.553,Z 1058.583,A -85,B 0,C 180,E1 21010.598,E2 21010.598} C_VEL
LIN {X 0,Y 460.481,Z 1072.612,A -85,B 0,C 180,E1 21008.548,E2 21008.548} C_VEL
LIN {X 0,Y 455.618,Z 1086.107,A -85,B 0,C 180,E1 21006.336,E2 21006.336} C_VEL
LIN {X 0,Y 451.032,Z 1098.994,A -85,B 0,C 180,E1 21003.962,E2 21003.962} C_VEL
LIN {X 0,Y 445.925,Z 1113.965,A -85,B 0,C 180,E1 21000.818,E2 21000.818} C_VEL
LIN {X 0,Y 441.749,Z 1126.754,A -85,B 0,C 180,E1 20997.645,E2 20997.645} C_VEL
LIN {X 0,Y 438.918,Z 1136.324,A -85,B 0,C 180,E1 20994.925,E2 20994.925} C_VEL
LIN {X 0,Y 436.583,Z 1145.11,A -85,B 0,C 180,E1 20992.061,E2 20992.061} C_VEL
LIN {X 0,Y 435.932,Z 1147.901,A -85,B 0,C 180,E1 20991.092,E2 20991.092} C_VEL
LIN {X 0,Y 434.333,Z 1150.493,A -85,B 0,C 180,E1 20990.149,E2 20990.149} C_VEL
LIN {X 0,Y 426.846,Z 1157.175,A -85,B 0,C 180,E1 20987.654,E2 20987.654} C_VEL
LIN {X 0,Y 425.765,Z 1159.058,A -85,B 0,C 180,E1 20986.807,E2 20986.807} C_VEL
LIN {X 0,Y 424.649,Z 1166.006,A -85,B 0,C 180,E1 20982.925,E2 20982.925} C_VEL
LIN {X 0,Y 424.206,Z 1170.174,A -85,B 0,C 180,E1 20979.847,E2 20979.847} C_VEL
LIN {X 0,Y 424.013,Z 1173.004,A -85,B 0,C 180,E1 20977.043,E2 20977.043} C_VEL
LIN {X 0,Y 423.942,Z 1174.856,A -85,B 0,C 180,E1 20974.328,E2 20974.328} C_VEL
LIN {X 0,Y 423.924,Z 1175.831,A -85,B 0,C 180,E1 20971.622,E2 20971.622} C_VEL
LIN {X 0,Y 423.924,Z 1175.934,A -85,B 0,C 180,E1 20968.919,E2 20968.919} C_VEL
LIN {X 0,Y 423.94,Z 1175.098,A -85,B 0,C 180,E1 20966.078,E2 20966.078} C_VEL
LIN {X 0,Y 423.998,Z 1173.407,A -85,B 0,C 180,E1 20963.365,E2 20963.365} C_VEL
LIN {X 0,Y 424.152,Z 1170.827,A -85,B 0,C 180,E1 20960.639,E2 20960.639} C_VEL
LIN {X 0,Y 424.502,Z 1167.231,A -85,B 0,C 180,E1 20957.827,E2 20957.827} C_VEL
LIN {X 0,Y 425.132,Z 1162.665,A -85,B 0,C 180,E1 20955.007,E2 20955.007} C_VEL
LIN {X 0,Y 426.183,Z 1156.929,A -85,B 0,C 180,E1 20952.101,E2 20952.101} C_VEL
LIN {X 0,Y 427.894,Z 1149.399,A -85,B 0,C 180,E1 20948.909,E2 20948.909} C_VEL
LIN {X 0,Y 430.793,Z 1138.666,A -85,B 0,C 180,E1 20945.159,E2 20945.159} C_VEL
LIN {X 0,Y 433.797,Z 1128.842,A -85,B 0,C 180,E1 20942.252,E2 20942.252} C_VEL
LIN {X 0,Y 437.358,Z 1118.217,A -85,B 0,C 180,E1 20939.501,E2 20939.501} C_VEL
LIN {X 0,Y 441.59,Z 1106.246,A -85,B 0,C 180,E1 20936.774,E2 20936.774} C_VEL
LIN {X 0,Y 447.935,Z 1089.104,A -85,B 0,C 180,E1 20933.417,E2 20933.417} C_VEL
LIN {X 0,Y 453.208,Z 1075.039,A -85,B 0,C 180,E1 20931.041,E2 20931.041} C_VEL
LIN {X 0,Y 458.752,Z 1060.298,A -85,B 0,C 180,E1 20928.836,E2 20928.836} C_VEL
LIN {X 0,Y 464.461,Z 1044.941,A -85,B 0,C 180,E1 20926.799,E2 20926.799} C_VEL
LIN {X 0,Y 471.49,Z 1025.735,A -85,B 0,C 180,E1 20924.559,E2 20924.559} C_VEL
LIN {X 0,Y 478.934,Z 1004.057,A -85,B 0,C 180,E1 20922.403,E2 20922.403} C_VEL
LIN {X 0,Y 484.69,Z 986.507,A -85,B 0,C 180,E1 20920.883,E2 20920.883} C_VEL
LIN {X 0,Y 490.143,Z 968.847,A -85,B 0,C 180,E1 20919.53,E2 20919.53} C_VEL
LIN {X 0,Y 495.722,Z 949.446,A -85,B 0,C 180,E1 20918.223,E2 20918.223} C_VEL
LIN {X 0,Y 502.132,Z 925.296,A -85,B 0,C 180,E1 20916.825,E2 20916.825} C_VEL
LIN {X 0,Y 507.932,Z 899.835,A -85,B 0,C 180,E1 20915.612,E2 20915.612} C_VEL
LIN {X 0,Y 512.015,Z 879.564,A -85,B 0,C 180,E1 20914.8,E2 20914.8} C_VEL
LIN {X 0,Y 515.65,Z 858.691,A -85,B 0,C 180,E1 20914.097,E2 20914.097} C_VEL
LIN {X 0,Y 518.882,Z 836.623,A -85,B 0,C 180,E1 20913.488,E2 20913.488} C_VEL
LIN {X 0,Y 522.008,Z 809.252,A -85,B 0,C 180,E1 20912.905,E2 20912.905} C_VEL
LIN {X 0,Y 524.925,Z 763.677,A -85,B 0,C 180,E1 20912.178,E2 20912.178} C_VEL
LIN {X 0,Y 537.946,Z 541.415,A -85,B 0,C 180,E1 20908.744,E2 20908.744} C_VEL
LIN {X 0,Y 541.395,Z 484.595,A -85,B 0,C 180,E1 20907.857,E2 20907.857} C_VEL
LIN {X 0,Y 532.463,Z 471.434,A -85,B 0,C 180,E1 20905.559,E2 20905.559} C_VEL
LIN {X 0,Y 524.983,Z 461.076,A -85,B 0,C 180,E1 20903.428,E2 20903.428} C_VEL
LIN {X 0,Y 518.212,Z 451.827,A -85,B 0,C 180,E1 20901.269,E2 20901.269} C_VEL
LIN {X 0,Y 513.982,Z 446.338,A -85,B 0,C 180,E1 20899.785,E2 20899.785} C_VEL
LIN {X 0,Y 510.33,Z 441.562,A -85,B 0,C 180,E1 20898.388,E2 20898.388} C_VEL
LIN {X 0,Y 506.691,Z 436.844,A -85,B 0,C 180,E1 20896.863,E2 20896.863} C_VEL
LIN {X 0,Y 503.023,Z 432.163,A -85,B 0,C 180,E1 20895.153,E2 20895.153} C_VEL
LIN {X 0,Y 498.932,Z 427.309,A -85,B 0,C 180,E1 20892.971,E2 20892.971} C_VEL
LIN {X 0,Y 497.834,Z 425.698,A -85,B 0,C 180,E1 20892.292,E2 20892.292} C_VEL
LIN {X 0,Y 494.534,Z 422.27,A -85,B 0,C 180,E1 20890.072,E2 20890.072} C_VEL
LIN {X 0,Y 493.15,Z 419.751,A -85,B 0,C 180,E1 20888.864,E2 20888.864} C_VEL
LIN {X 0,Y 489.591,Z 416.463,A -85,B 0,C 180,E1 20884.921,E2 20884.921} C_VEL
LIN {X 0,Y 488.675,Z 413.531,A -85,B 0,C 180,E1 20882.463,E2 20882.463} C_VEL
LIN {X 0,Y 488.795,Z 413.798,A -85,B 0,C 180,E1 20877.538,E2 20877.538} C_VEL
LIN {X 0,Y 490.8,Z 418.111,A -85,B 0,C 180,E1 20873.801,E2 20873.801} C_VEL
LIN {X 0,Y 493.562,Z 420.216,A -85,B 0,C 180,E1 20871.202,E2 20871.202} C_VEL
LIN {X 0,Y 496.282,Z 424.458,A -85,B 0,C 180,E1 20869.083,E2 20869.083} C_VEL
LIN {X 0,Y 498.406,Z 426.318,A -85,B 0,C 180,E1 20867.781,E2 20867.781} C_VEL
LIN {X 0,Y 501.689,Z 430.732,A -85,B 0,C 180,E1 20865.927,E2 20865.927} C_VEL
LIN {X 0,Y 503.255,Z 432.471,A -85,B 0,C 180,E1 20865.149,E2 20865.149} C_VEL
LIN {X 0,Y 508.343,Z 439.048,A -85,B 0,C 180,E1 20862.84,E2 20862.84} C_VEL
LIN {X 0,Y 514.412,Z 447.785,A -85,B 0,C 180,E1 20860.439,E2 20860.439} C_VEL
LIN {X 0,Y 520.269,Z 456.269,A -85,B 0,C 180,E1 20858.405,E2 20858.405} C_VEL
LIN {X 0,Y 529.163,Z 469.839,A -85,B 0,C 180,E1 20855.674,E2 20855.674} C_VEL
LIN {X 0,Y 538.388,Z 484.748,A -85,B 0,C 180,E1 20853.173,E2 20853.173} C_VEL
LIN {X 0,Y 541.467,Z 490.306,A -85,B 0,C 180,E1 20852.386,E2 20852.386} C_VEL
LIN {X 0,Y 528.873,Z 702.716,A -85,B 0,C 180,E1 20849.095,E2 20849.095} C_VEL
LIN {X 0,Y 521.937,Z 821.707,A -85,B 0,C 180,E1 20847.243,E2 20847.243} C_VEL
LIN {X 0,Y 519.139,Z 849.212,A -85,B 0,C 180,E1 20846.72,E2 20846.72} C_VEL
LIN {X 0,Y 515.193,Z 875.783,A -85,B 0,C 180,E1 20846.04,E2 20846.04} C_VEL
LIN {X 0,Y 511.407,Z 897.246,A -85,B 0,C 180,E1 20845.35,E2 20845.35} C_VEL
LIN {X 0,Y 507.253,Z 917.745,A -85,B 0,C 180,E1 20844.561,E2 20844.561} C_VEL
LIN {X 0,Y 502.486,Z 938.723,A -85,B 0,C 180,E1 20843.608,E2 20843.608} C_VEL
LIN {X 0,Y 496.214,Z 963.652,A -85,B 0,C 180,E1 20842.267,E2 20842.267} C_VEL
LIN {X 0,Y 489.681,Z 986.58,A -85,B 0,C 180,E1 20840.794,E2 20840.794} C_VEL
LIN {X 0,Y 483.917,Z 1005.519,A -85,B 0,C 180,E1 20839.393,E2 20839.393} C_VEL
LIN {X 0,Y 478.027,Z 1023.859,A -85,B 0,C 180,E1 20837.849,E2 20837.849} C_VEL
LIN {X 0,Y 471.225,Z 1044.2,A -85,B 0,C 180,E1 20835.894,E2 20835.894} C_VEL
LIN {X 0,Y 463.647,Z 1065.822,A -85,B 0,C 180,E1 20833.466,E2 20833.466} C_VEL
LIN {X 0,Y 457.781,Z 1082.204,A -85,B 0,C 180,E1 20831.353,E2 20831.353} C_VEL
LIN {X 0,Y 452.456,Z 1097.041,A -85,B 0,C 180,E1 20829.199,E2 20829.199} C_VEL
LIN {X 0,Y 447.239,Z 1111.68,A -85,B 0,C 180,E1 20826.809,E2 20826.809} C_VEL
LIN {X 0,Y 441.216,Z 1128.987,A -85,B 0,C 180,E1 20823.569,E2 20823.569} C_VEL
LIN {X 0,Y 436.699,Z 1142.644,A -85,B 0,C 180,E1 20820.58,E2 20820.58} C_VEL
LIN {X 0,Y 433.356,Z 1153.421,A -85,B 0,C 180,E1 20817.907,E2 20817.907} C_VEL
LIN {X 0,Y 430.508,Z 1163.506,A -85,B 0,C 180,E1 20815.067,E2 20815.067} C_VEL
LIN {X 0,Y 427.837,Z 1174.397,A -85,B 0,C 180,E1 20811.525,E2 20811.525} C_VEL
LIN {X 0,Y 426.007,Z 1183.138,A -85,B 0,C 180,E1 20808.048,E2 20808.048} C_VEL
LIN {X 0,Y 425.026,Z 1189.276,A -85,B 0,C 180,E1 20805.137,E2 20805.137} C_VEL
LIN {X 0,Y 424.431,Z 1194.089,A -85,B 0,C 180,E1 20802.379,E2 20802.379} C_VEL
LIN {X 0,Y 424.117,Z 1197.917,A -85,B 0,C 180,E1 20799.636,E2 20799.636} C_VEL
LIN {X 0,Y 423.973,Z 1200.782,A -85,B 0,C 180,E1 20796.908,E2 20796.908} C_VEL
LIN {X 0,Y 423.929,Z 1202.7,A -85,B 0,C 180,E1 20794.193,E2 20794.193} C_VEL
LIN {X 0,Y 423.927,Z 1203.68,A -85,B 0,C 180,E1 20791.487,E2 20791.487} C_VEL
LIN {X 0,Y 423.927,Z 1203.75,A -85,B 0,C 180,E1 20788.919,E2 20788.919} C_VEL
LIN {X 0,Y 423.927,Z 1202.91,A -85,B 0,C 180,E1 20786.213,E2 20786.213} C_VEL
LIN {X 0,Y 423.966,Z 1201.133,A -85,B 0,C 180,E1 20783.5,E2 20783.5} C_VEL
LIN {X 0,Y 424.086,Z 1198.411,A -85,B 0,C 180,E1 20780.774,E2 20780.774} C_VEL
LIN {X 0,Y 424.368,Z 1194.728,A -85,B 0,C 180,E1 20778.034,E2 20778.034} C_VEL
LIN {X 0,Y 424.953,Z 1189.8,A -85,B 0,C 180,E1 20775.14,E2 20775.14} C_VEL
LIN {X 0,Y 425.847,Z 1184.073,A -85,B 0,C 180,E1 20772.369,E2 20772.369} C_VEL
LIN {X 0,Y 427.276,Z 1176.81,A -85,B 0,C 180,E1 20769.401,E2 20769.401} C_VEL
LIN {X 0,Y 429.755,Z 1166.518,A -85,B 0,C 180,E1 20765.828,E2 20765.828} C_VEL
LIN {X 0,Y 432.917,Z 1154.923,A -85,B 0,C 180,E1 20762.488,E2 20762.488} C_VEL
LIN {X 0,Y 436.289,Z 1143.934,A -85,B 0,C 180,E1 20759.723,E2 20759.723} C_VEL
LIN {X 0,Y 440.102,Z 1132.22,A -85,B 0,C 180,E1 20757.114,E2 20757.114} C_VEL
LIN {X 0,Y 444.84,Z 1118.44,A -85,B 0,C 180,E1 20754.398,E2 20754.398} C_VEL
LIN {X 0,Y 451.552,Z 1099.596,A -85,B 0,C 180,E1 20751.198,E2 20751.198} C_VEL
LIN {X 0,Y 457.103,Z 1084.082,A -85,B 0,C 180,E1 20748.91,E2 20748.91} C_VEL
LIN {X 0,Y 462.546,Z 1068.871,A -85,B 0,C 180,E1 20746.916,E2 20746.916} C_VEL
LIN {X 0,Y 468.251,Z 1052.687,A -85,B 0,C 180,E1 20745.026,E2 20745.026} C_VEL
LIN {X 0,Y 474.828,Z 1033.576,A -85,B 0,C 180,E1 20743.056,E2 20743.056} C_VEL
LIN {X 0,Y 482.569,Z 1009.797,A -85,B 0,C 180,E1 20740.955,E2 20740.955} C_VEL
LIN {X 0,Y 488.468,Z 990.58,A -85,B 0,C 180,E1 20739.494,E2 20739.494} C_VEL
LIN {X 0,Y 493.761,Z 972.169,A -85,B 0,C 180,E1 20738.262,E2 20738.262} C_VEL
LIN {X 0,Y 499.005,Z 952.51,A -85,B 0,C 180,E1 20737.111,E2 20737.111} C_VEL
LIN {X 0,Y 504.057,Z 931.874,A -85,B 0,C 180,E1 20736.068,E2 20736.068} C_VEL
LIN {X 0,Y 509.901,Z 904.983,A -85,B 0,C 180,E1 20734.932,E2 20734.932} C_VEL
LIN {X 0,Y 514.336,Z 880.663,A -85,B 0,C 180,E1 20734.111,E2 20734.111} C_VEL
LIN {X 0,Y 517.662,Z 859.059,A -85,B 0,C 180,E1 20733.518,E2 20733.518} C_VEL
LIN {X 0,Y 520.44,Z 837.001,A -85,B 0,C 180,E1 20733.04,E2 20733.04} C_VEL
LIN {X 0,Y 522.775,Z 809.577,A -85,B 0,C 180,E1 20732.557,E2 20732.557} C_VEL
LIN {X 0,Y 535.621,Z 585.923,A -85,B 0,C 180,E1 20729.104,E2 20729.104} C_VEL
LIN {X 0,Y 541.318,Z 489.808,A -85,B 0,C 180,E1 20727.592,E2 20727.592} C_VEL
LIN {X 0,Y 532.02,Z 474.49,A -85,B 0,C 180,E1 20725.165,E2 20725.165} C_VEL
LIN {X 0,Y 524.134,Z 462.252,A -85,B 0,C 180,E1 20722.871,E2 20722.871} C_VEL
LIN {X 0,Y 516.441,Z 450.636,A -85,B 0,C 180,E1 20720.337,E2 20720.337} C_VEL
LIN {X 0,Y 509.24,Z 440.338,A -85,B 0,C 180,E1 20717.601,E2 20717.601} C_VEL
LIN {X 0,Y 506.159,Z 436.369,A -85,B 0,C 180,E1 20716.291,E2 20716.291} C_VEL
LIN {X 0,Y 502.195,Z 431.225,A -85,B 0,C 180,E1 20714.411,E2 20714.411} C_VEL
LIN {X 0,Y 498.682,Z 426.901,A -85,B 0,C 180,E1 20712.506,E2 20712.506} C_VEL
LIN {X 0,Y 497.748,Z 425.677,A -85,B 0,C 180,E1 20711.941,E2 20711.941} C_VEL
LIN {X 0,Y 494.653,Z 422.426,A -85,B 0,C 180,E1 20709.894,E2 20709.894} C_VEL
LIN {X 0,Y 493.159,Z 419.753,A -85,B 0,C 180,E1 20708.629,E2 20708.629} C_VEL
LIN {X 0,Y 489.631,Z 416.567,A -85,B 0,C 180,E1 20704.92,E2 20704.92} C_VEL
LIN {X 0,Y 488.559,Z 413.522,A -85,B 0,C 180,E1 20702.463,E2 20702.463} C_VEL
LIN {X 0,Y 488.682,Z 413.611,A -85,B 0,C 180,E1 20696.716,E2 20696.716} C_VEL
LIN {X 0,Y 489.841,Z 416.885,A -85,B 0,C 180,E1 20694.26,E2 20694.26} C_VEL
LIN {X 0,Y 493.448,Z 420.198,A -85,B 0,C 180,E1 20690.612,E2 20690.612} C_VEL
LIN {X 0,Y 495.703,Z 423.862,A -85,B 0,C 180,E1 20688.834,E2 20688.834} C_VEL
LIN {X 0,Y 498.352,Z 426.357,A -85,B 0,C 180,E1 20687.191,E2 20687.191} C_VEL
LIN {X 0,Y 501.555,Z 430.716,A -85,B 0,C 180,E1 20685.393,E2 20685.393} C_VEL
LIN {X 0,Y 503.134,Z 432.417,A -85,B 0,C 180,E1 20684.615,E2 20684.615} C_VEL
LIN {X 0,Y 506.992,Z 437.133,A -85,B 0,C 180,E1 20682.852,E2 20682.852} C_VEL
LIN {X 0,Y 512.481,Z 444.402,A -85,B 0,C 180,E1 20680.629,E2 20680.629} C_VEL
LIN {X 0,Y 517.152,Z 450.517,A -85,B 0,C 180,E1 20678.953,E2 20678.953} C_VEL
LIN {X 0,Y 523.109,Z 458.43,A -85,B 0,C 180,E1 20677.02,E2 20677.02} C_VEL
LIN {X 0,Y 531.718,Z 470.467,A -85,B 0,C 180,E1 20674.522,E2 20674.522} C_VEL
LIN {X 0,Y 540.217,Z 482.927,A -85,B 0,C 180,E1 20672.317,E2 20672.317} C_VEL
LIN {X 0,Y 541.333,Z 484.861,A -85,B 0,C 180,E1 20672.036,E2 20672.036} C_VEL
LIN {X 0,Y 528.408,Z 701.393,A -85,B 0,C 180,E1 20668.689,E2 20668.689} C_VEL
LIN {X 0,Y 522.382,Z 803.452,A -85,B 0,C 180,E1 20667.098,E2 20667.098} C_VEL
LIN {X 0,Y 519.628,Z 830.817,A -85,B 0,C 180,E1 20666.563,E2 20666.563} C_VEL
LIN {X 0,Y 515.884,Z 856.9,A -85,B 0,C 180,E1 20665.864,E2 20665.864} C_VEL
LIN {X 0,Y 512.246,Z 878.006,A -85,B 0,C 180,E1 20665.163,E2 20665.163} C_VEL
LIN {X 0,Y 508.167,Z 898.474,A -85,B 0,C 180,E1 20664.351,E2 20664.351} C_VEL
LIN {X 0,Y 503.132,Z 920.782,A -85,B 0,C 180,E1 20663.308,E2 20663.308} C_VEL
LIN {X 0,Y 496.209,Z 947.586,A -85,B 0,C 180,E1 20661.799,E2 20661.799} C_VEL
LIN {X 0,Y 490.59,Z 967.233,A -85,B 0,C 180,E1 20660.49,E2 20660.49} C_VEL
LIN {X 0,Y 485.137,Z 984.965,A -85,B 0,C 180,E1 20659.146,E2 20659.146} C_VEL
LIN {X 0,Y 479.434,Z 1002.417,A -85,B 0,C 180,E1 20657.651,E2 20657.651} C_VEL
LIN {X 0,Y 473.095,Z 1020.937,A -85,B 0,C 180,E1 20655.849,E2 20655.849} C_VEL
LIN {X 0,Y 465.224,Z 1042.87,A -85,B 0,C 180,E1 20653.367,E2 20653.367} C_VEL
LIN {X 0,Y 459.104,Z 1059.315,A -85,B 0,C 180,E1 20651.208,E2 20651.208} C_VEL
LIN {X 0,Y 453.684,Z 1073.72,A -85,B 0,C 180,E1 20649.072,E2 20649.072} C_VEL
LIN {X 0,Y 448.367,Z 1087.898,A -85,B 0,C 180,E1 20646.701,E2 20646.701} C_VEL
LIN {X 0,Y 442.43,Z 1104.006,A -85,B 0,C 180,E1 20643.62,E2 20643.62} C_VEL
LIN {X 0,Y 437.489,Z 1117.846,A -85,B 0,C 180,E1 20640.498,E2 20640.498} C_VEL
LIN {X 0,Y 433.926,Z 1128.447,A -85,B 0,C 180,E1 20637.767,E2 20637.767} C_VEL
LIN {X 0,Y 430.898,Z 1138.301,A -85,B 0,C 180,E1 20634.863,E2 20634.863} C_VEL
LIN {X 0,Y 428.051,Z 1148.834,A -85,B 0,C 180,E1 20631.226,E2 20631.226} C_VEL
LIN {X 0,Y 426.222,Z 1156.739,A -85,B 0,C 180,E1 20627.897,E2 20627.897} C_VEL
LIN {X 0,Y 425.765,Z 1159.058,A -85,B 0,C 180,E1 20626.807,E2 20626.807} C_VEL
LIN {X 0,Y 424.427,Z 1161.168,A -85,B 0,C 180,E1 20625.816,E2 20625.816} C_VEL
LIN {X 0,Y 417.342,Z 1166.362,A -85,B 0,C 180,E1 20623.092,E2 20623.092} C_VEL
LIN {X 0,Y 416.548,Z 1167.561,A -85,B 0,C 180,E1 20622.274,E2 20622.274} C_VEL
LIN {X 0,Y 416.165,Z 1171.299,A -85,B 0,C 180,E1 20619.263,E2 20619.263} C_VEL
LIN {X 0,Y 415.993,Z 1174.148,A -85,B 0,C 180,E1 20616.071,E2 20616.071} C_VEL
LIN {X 0,Y 415.932,Z 1175.965,A -85,B 0,C 180,E1 20612.48,E2 20612.48} C_VEL
LIN {X 0,Y 415.924,Z 1176.241,A -85,B 0,C 180,E1 20609.174,E2 20609.174} C_VEL
LIN {X 0,Y 415.943,Z 1175.493,A -85,B 0,C 180,E1 20606.279,E2 20606.279} C_VEL
LIN {X 0,Y 416.006,Z 1173.781,A -85,B 0,C 180,E1 20603.375,E2 20603.375} C_VEL
LIN {X 0,Y 416.179,Z 1171.092,A -85,B 0,C 180,E1 20600.458,E2 20600.458} C_VEL
LIN {X 0,Y 416.546,Z 1167.603,A -85,B 0,C 180,E1 20597.665,E2 20597.665} C_VEL
LIN {X 0,Y 417.197,Z 1163.179,A -85,B 0,C 180,E1 20594.857,E2 20594.857} C_VEL
LIN {X 0,Y 418.301,Z 1157.492,A -85,B 0,C 180,E1 20591.896,E2 20591.896} C_VEL
LIN {X 0,Y 419.909,Z 1150.7,A -85,B 0,C 180,E1 20588.928,E2 20588.928} C_VEL
LIN {X 0,Y 422.623,Z 1141.163,A -85,B 0,C 180,E1 20585.393,E2 20585.393} C_VEL
LIN {X 0,Y 426.274,Z 1129.617,A -85,B 0,C 180,E1 20581.871,E2 20581.871} C_VEL
LIN {X 0,Y 429.988,Z 1119.05,A -85,B 0,C 180,E1 20579.077,E2 20579.077} C_VEL
LIN {X 0,Y 434.147,Z 1107.762,A -85,B 0,C 180,E1 20576.446,E2 20576.446} C_VEL
LIN {X 0,Y 439.837,Z 1093.075,A -85,B 0,C 180,E1 20573.445,E2 20573.445} C_VEL
LIN {X 0,Y 446.439,Z 1076.141,A -85,B 0,C 180,E1 20570.502,E2 20570.502} C_VEL
LIN {X 0,Y 452.348,Z 1061.024,A -85,B 0,C 180,E1 20568.208,E2 20568.208} C_VEL
LIN {X 0,Y 458.066,Z 1046.21,A -85,B 0,C 180,E1 20566.216,E2 20566.216} C_VEL
LIN {X 0,Y 464.04,Z 1030.386,A -85,B 0,C 180,E1 20564.328,E2 20564.328} C_VEL
LIN {X 0,Y 471.564,Z 1009.857,A -85,B 0,C 180,E1 20562.18,E2 20562.18} C_VEL
LIN {X 0,Y 478.891,Z 988.226,A -85,B 0,C 180,E1 20560.261,E2 20560.261} C_VEL
LIN {X 0,Y 484.8,Z 969.711,A -85,B 0,C 180,E1 20558.829,E2 20558.829} C_VEL
LIN {X 0,Y 490.468,Z 950.6,A -85,B 0,C 180,E1 20557.533,E2 20557.533} C_VEL
LIN {X 0,Y 496.229,Z 929.546,A -85,B 0,C 180,E1 20556.297,E2 20556.297} C_VEL
LIN {X 0,Y 502.725,Z 902.644,A -85,B 0,C 180,E1 20554.974,E2 20554.974} C_VEL
LIN {X 0,Y 507.333,Z 880.48,A -85,B 0,C 180,E1 20554.078,E2 20554.078} C_VEL
LIN {X 0,Y 511.095,Z 859.505,A -85,B 0,C 180,E1 20553.368,E2 20553.368} C_VEL
LIN {X 0,Y 514.353,Z 837.911,A -85,B 0,C 180,E1 20552.769,E2 20552.769} C_VEL
LIN {X 0,Y 517.436,Z 812.256,A -85,B 0,C 180,E1 20552.211,E2 20552.211} C_VEL
LIN {X 0,Y 520.157,Z 773.303,A -85,B 0,C 180,E1 20551.578,E2 20551.578} C_VEL
LIN {X 0,Y 533.581,Z 550.612,A -85,B 0,C 180,E1 20548.13,E2 20548.13} C_VEL
LIN {X 0,Y 537.363,Z 489.299,A -85,B 0,C 180,E1 20547.161,E2 20547.161} C_VEL
LIN {X 0,Y 528.729,Z 476.521,A -85,B 0,C 180,E1 20544.854,E2 20544.854} C_VEL
LIN {X 0,Y 520.583,Z 464.989,A -85,B 0,C 180,E1 20542.412,E2 20542.412} C_VEL
LIN {X 0,Y 513.158,Z 454.925,A -85,B 0,C 180,E1 20539.878,E2 20539.878} C_VEL
LIN {X 0,Y 508.539,Z 448.952,A -85,B 0,C 180,E1 20538.099,E2 20538.099} C_VEL
LIN {X 0,Y 504.963,Z 444.291,A -85,B 0,C 180,E1 20536.567,E2 20536.567} C_VEL
LIN {X 0,Y 500.82,Z 439.006,A -85,B 0,C 180,E1 20534.57,E2 20534.57} C_VEL
LIN {X 0,Y 497.482,Z 434.854,A -85,B 0,C 180,E1 20532.714,E2 20532.714} C_VEL
LIN {X 0,Y 496.49,Z 433.44,A -85,B 0,C 180,E1 20532.09,E2 20532.09} C_VEL
LIN {X 0,Y 493.265,Z 429.961,A -85,B 0,C 180,E1 20529.863,E2 20529.863} C_VEL
LIN {X 0,Y 492.043,Z 427.64,A -85,B 0,C 180,E1 20528.767,E2 20528.767} C_VEL
LIN {X 0,Y 488.546,Z 424.341,A -85,B 0,C 180,E1 20524.814,E2 20524.814} C_VEL
LIN {X 0,Y 487.701,Z 421.471,A -85,B 0,C 180,E1 20522.468,E2 20522.468} C_VEL
LIN {X 0,Y 487.781,Z 421.688,A -85,B 0,C 180,E1 20517.65,E2 20517.65} C_VEL
LIN {X 0,Y 489.727,Z 425.992,A -85,B 0,C 180,E1 20513.905,E2 20513.905} C_VEL
LIN {X 0,Y 492.378,Z 428.049,A -85,B 0,C 180,E1 20511.357,E2 20511.357} C_VEL
LIN {X 0,Y 495.139,Z 432.344,A -85,B 0,C 180,E1 20509.175,E2 20509.175} C_VEL
LIN {X 0,Y 497.14,Z 434.19,A -85,B 0,C 180,E1 20507.926,E2 20507.926} C_VEL
LIN {X 0,Y 500.501,Z 438.638,A -85,B 0,C 180,E1 20506.011,E2 20506.011} C_VEL
LIN {X 0,Y 501.929,Z 440.377,A -85,B 0,C 180,E1 20505.286,E2 20505.286} C_VEL
LIN {X 0,Y 506.716,Z 446.595,A -85,B 0,C 180,E1 20503.079,E2 20503.079} C_VEL
LIN {X 0,Y 512.622,Z 455.255,A -85,B 0,C 180,E1 20500.694,E2 20500.694} C_VEL
LIN {X 0,Y 518.395,Z 463.778,A -85,B 0,C 180,E1 20498.65,E2 20498.65} C_VEL
LIN {X 0,Y 527.002,Z 477.148,A -85,B 0,C 180,E1 20495.955,E2 20495.955} C_VEL
LIN {X 0,Y 536.496,Z 492.704,A -85,B 0,C 180,E1 20493.34,E2 20493.34} C_VEL
LIN {X 0,Y 537.484,Z 494.703,A -85,B 0,C 180,E1 20493.075,E2 20493.075} C_VEL
LIN {X 0,Y 524.403,Z 708.85,A -85,B 0,C 180,E1 20489.751,E2 20489.751} C_VEL
LIN {X 0,Y 517.617,Z 821.569,A -85,B 0,C 180,E1 20487.991,E2 20487.991} C_VEL
LIN {X 0,Y 514.723,Z 849.235,A -85,B 0,C 180,E1 20487.464,E2 20487.464} C_VEL
LIN {X 0,Y 510.699,Z 875.636,A -85,B 0,C 180,E1 20486.789,E2 20486.789} C_VEL
LIN {X 0,Y 506.831,Z 897.03,A -85,B 0,C 180,E1 20486.103,E2 20486.103} C_VEL
LIN {X 0,Y 502.578,Z 917.456,A -85,B 0,C 180,E1 20485.319,E2 20485.319} C_VEL
LIN {X 0,Y 497.652,Z 938.568,A -85,B 0,C 180,E1 20484.361,E2 20484.361} C_VEL
LIN {X 0,Y 490.955,Z 964.294,A -85,B 0,C 180,E1 20482.971,E2 20482.971} C_VEL
LIN {X 0,Y 484.491,Z 986.313,A -85,B 0,C 180,E1 20481.553,E2 20481.553} C_VEL
LIN {X 0,Y 478.343,Z 1005.901,A -85,B 0,C 180,E1 20480.096,E2 20480.096} C_VEL
LIN {X 0,Y 472.271,Z 1024.196,A -85,B 0,C 180,E1 20478.544,E2 20478.544} C_VEL
LIN {X 0,Y 464.847,Z 1045.671,A -85,B 0,C 180,E1 20476.458,E2 20476.458} C_VEL
LIN {X 0,Y 457.189,Z 1066.575,A -85,B 0,C 180,E1 20474.063,E2 20474.063} C_VEL
LIN {X 0,Y 451.301,Z 1082.399,A -85,B 0,C 180,E1 20471.996,E2 20471.996} C_VEL
LIN {X 0,Y 445.615,Z 1097.624,A -85,B 0,C 180,E1 20469.753,E2 20469.753} C_VEL
LIN {X 0,Y 439.39,Z 1114.539,A -85,B 0,C 180,E1 20466.923,E2 20466.923} C_VEL
LIN {X 0,Y 433.481,Z 1130.653,A -85,B 0,C 180,E1 20463.772,E2 20463.772} C_VEL
LIN {X 0,Y 429.207,Z 1143.077,A -85,B 0,C 180,E1 20460.985,E2 20460.985} C_VEL
LIN {X 0,Y 425.633,Z 1154.122,A -85,B 0,C 180,E1 20458.175,E2 20458.175} C_VEL
LIN {X 0,Y 422.129,Z 1166.243,A -85,B 0,C 180,E1 20454.637,E2 20454.637} C_VEL
LIN {X 0,Y 419.555,Z 1176.303,A -85,B 0,C 180,E1 20451.091,E2 20451.091} C_VEL
LIN {X 0,Y 418.032,Z 1183.491,A -85,B 0,C 180,E1 20448.116,E2 20448.116} C_VEL
LIN {X 0,Y 417.027,Z 1189.531,A -85,B 0,C 180,E1 20445.149,E2 20445.149} C_VEL
LIN {X 0,Y 416.407,Z 1194.414,A -85,B 0,C 180,E1 20442.229,E2 20442.229} C_VEL
LIN {X 0,Y 416.088,Z 1198.311,A -85,B 0,C 180,E1 20439.265,E2 20439.265} C_VEL
LIN {X 0,Y 415.955,Z 1201.339,A -85,B 0,C 180,E1 20436.071,E2 20436.071} C_VEL
LIN {X 0,Y 415.929,Z 1203.251,A -85,B 0,C 180,E1 20432.48,E2 20432.48} C_VEL
LIN {X 0,Y 415.923,Z 1203.534,A -85,B 0,C 180,E1 20429.174,E2 20429.174} C_VEL
LIN {X 0,Y 415.93,Z 1202.717,A -85,B 0,C 180,E1 20426.279,E2 20426.279} C_VEL
LIN {X 0,Y 415.97,Z 1200.869,A -85,B 0,C 180,E1 20423.375,E2 20423.375} C_VEL
LIN {X 0,Y 416.099,Z 1198.145,A -85,B 0,C 180,E1 20420.596,E2 20420.596} C_VEL
LIN {X 0,Y 416.407,Z 1194.414,A -85,B 0,C 180,E1 20417.771,E2 20417.771} C_VEL
LIN {X 0,Y 417.027,Z 1189.531,A -85,B 0,C 180,E1 20414.851,E2 20414.851} C_VEL
LIN {X 0,Y 418.032,Z 1183.489,A -85,B 0,C 180,E1 20411.884,E2 20411.884} C_VEL
LIN {X 0,Y 419.557,Z 1176.3,A -85,B 0,C 180,E1 20408.909,E2 20408.909} C_VEL
LIN {X 0,Y 422.247,Z 1165.779,A -85,B 0,C 180,E1 20405.221,E2 20405.221} C_VEL
LIN {X 0,Y 425.635,Z 1154.124,A -85,B 0,C 180,E1 20401.825,E2 20401.825} C_VEL
LIN {X 0,Y 429.208,Z 1143.07,A -85,B 0,C 180,E1 20399.014,E2 20399.014} C_VEL
LIN {X 0,Y 433.479,Z 1130.645,A -85,B 0,C 180,E1 20396.228,E2 20396.228} C_VEL
LIN {X 0,Y 439.587,Z 1113.948,A -85,B 0,C 180,E1 20392.977,E2 20392.977} C_VEL
LIN {X 0,Y 445.611,Z 1097.598,A -85,B 0,C 180,E1 20390.247,E2 20390.247} C_VEL
LIN {X 0,Y 451.296,Z 1082.367,A -85,B 0,C 180,E1 20388.003,E2 20388.003} C_VEL
LIN {X 0,Y 457.374,Z 1066.022,A -85,B 0,C 180,E1 20385.872,E2 20385.872} C_VEL
LIN {X 0,Y 465.255,Z 1044.38,A -85,B 0,C 180,E1 20383.416,E2 20383.416} C_VEL
LIN {X 0,Y 472.261,Z 1024.119,A -85,B 0,C 180,E1 20381.455,E2 20381.455} C_VEL
LIN {X 0,Y 478.482,Z 1005.339,A -85,B 0,C 180,E1 20379.865,E2 20379.865} C_VEL
LIN {X 0,Y 484.77,Z 985.259,A -85,B 0,C 180,E1 20378.378,E2 20378.378} C_VEL
LIN {X 0,Y 491.985,Z 960.336,A -85,B 0,C 180,E1 20376.801,E2 20376.801} C_VEL
LIN {X 0,Y 497.909,Z 937.288,A -85,B 0,C 180,E1 20375.582,E2 20375.582} C_VEL
LIN {X 0,Y 502.698,Z 916.657,A -85,B 0,C 180,E1 20374.653,E2 20374.653} C_VEL
LIN {X 0,Y 506.964,Z 896.069,A -85,B 0,C 180,E1 20373.869,E2 20373.869} C_VEL
LIN {X 0,Y 510.982,Z 873.635,A -85,B 0,C 180,E1 20373.157,E2 20373.157} C_VEL
LIN {X 0,Y 515.197,Z 844.539,A -85,B 0,C 180,E1 20372.445,E2 20372.445} C_VEL
LIN {X 0,Y 517.646,Z 820.316,A -85,B 0,C 180,E1 20371.993,E2 20371.993} C_VEL
LIN {X 0,Y 530.056,Z 613.199,A -85,B 0,C 180,E1 20368.771,E2 20368.771} C_VEL
LIN {X 0,Y 537.376,Z 494.34,A -85,B 0,C 180,E1 20366.916,E2 20366.916} C_VEL
LIN {X 0,Y 527.596,Z 478.214,A -85,B 0,C 180,E1 20364.254,E2 20364.254} C_VEL
LIN {X 0,Y 519.221,Z 465.121,A -85,B 0,C 180,E1 20361.67,E2 20361.67} C_VEL
LIN {X 0,Y 513.062,Z 455.993,A -85,B 0,C 180,E1 20359.526,E2 20359.526} C_VEL
LIN {X 0,Y 507.334,Z 447.535,A -85,B 0,C 180,E1 20357.255,E2 20357.255} C_VEL
LIN {X 0,Y 504.437,Z 443.79,A -85,B 0,C 180,E1 20355.993,E2 20355.993} C_VEL
LIN {X 0,Y 500.776,Z 438.925,A -85,B 0,C 180,E1 20354.217,E2 20354.217} C_VEL
LIN {X 0,Y 497.231,Z 434.443,A -85,B 0,C 180,E1 20352.249,E2 20352.249} C_VEL
LIN {X 0,Y 496.399,Z 433.423,A -85,B 0,C 180,E1 20351.738,E2 20351.738} C_VEL
LIN {X 0,Y 493.303,Z 429.995,A -85,B 0,C 180,E1 20349.626,E2 20349.626} C_VEL
LIN {X 0,Y 492.047,Z 427.645,A -85,B 0,C 180,E1 20348.531,E2 20348.531} C_VEL
LIN {X 0,Y 488.577,Z 424.446,A -85,B 0,C 180,E1 20344.813,E2 20344.813} C_VEL
LIN {X 0,Y 487.585,Z 421.463,A -85,B 0,C 180,E1 20342.468,E2 20342.468} C_VEL
LIN {X 0,Y 487.663,Z 421.508,A -85,B 0,C 180,E1 20336.826,E2 20336.826} C_VEL
LIN {X 0,Y 488.784,Z 424.764,A -85,B 0,C 180,E1 20334.365,E2 20334.365} C_VEL
LIN {X 0,Y 492.262,Z 428.04,A -85,B 0,C 180,E1 20330.766,E2 20330.766} C_VEL
LIN {X 0,Y 494.731,Z 431.931,A -85,B 0,C 180,E1 20328.812,E2 20328.812} C_VEL
LIN {X 0,Y 497.084,Z 434.238,A -85,B 0,C 180,E1 20327.335,E2 20327.335} C_VEL
LIN {X 0,Y 500.368,Z 438.623,A -85,B 0,C 180,E1 20325.476,E2 20325.476} C_VEL
LIN {X 0,Y 501.808,Z 440.322,A -85,B 0,C 180,E1 20324.751,E2 20324.751} C_VEL
LIN {X 0,Y 506.374,Z 446.138,A -85,B 0,C 180,E1 20322.652,E2 20322.652} C_VEL
LIN {X 0,Y 510.791,Z 451.964,A -85,B 0,C 180,E1 20320.859,E2 20320.859} C_VEL
LIN {X 0,Y 517.271,Z 460.437,A -85,B 0,C 180,E1 20318.542,E2 20318.542} C_VEL
LIN {X 0,Y 527.565,Z 474.804,A -85,B 0,C 180,E1 20315.357,E2 20315.357} C_VEL
LIN {X 0,Y 537.151,Z 489.054,A -85,B 0,C 180,E1 20312.777,E2 20312.777} C_VEL
LIN {X 0,Y 537.326,Z 489.805,A -85,B 0,C 180,E1 20312.718,E2 20312.718} C_VEL
LIN {X 0,Y 524.036,Z 705.995,A -85,B 0,C 180,E1 20309.37,E2 20309.37} C_VEL
LIN {X 0,Y 518.077,Z 803.738,A -85,B 0,C 180,E1 20307.841,E2 20307.841} C_VEL
LIN {X 0,Y 515.255,Z 831.094,A -85,B 0,C 180,E1 20307.306,E2 20307.306} C_VEL
LIN {X 0,Y 511.42,Z 857.175,A -85,B 0,C 180,E1 20306.609,E2 20306.609} C_VEL
LIN {X 0,Y 507.688,Z 878.281,A -85,B 0,C 180,E1 20305.909,E2 20305.909} C_VEL
LIN {X 0,Y 503.506,Z 898.748,A -85,B 0,C 180,E1 20305.098,E2 20305.098} C_VEL
LIN {X 0,Y 498.599,Z 919.934,A -85,B 0,C 180,E1 20304.111,E2 20304.111} C_VEL
LIN {X 0,Y 491.752,Z 946.074,A -85,B 0,C 180,E1 20302.655,E2 20302.655} C_VEL
LIN {X 0,Y 485.664,Z 966.783,A -85,B 0,C 180,E1 20301.284,E2 20301.284} C_VEL
LIN {X 0,Y 480,Z 984.668,A -85,B 0,C 180,E1 20299.933,E2 20299.933} C_VEL
LIN {X 0,Y 474.202,Z 1001.876,A -85,B 0,C 180,E1 20298.462,E2 20298.462} C_VEL
LIN {X 0,Y 468.009,Z 1019.41,A -85,B 0,C 180,E1 20296.762,E2 20296.762} C_VEL
LIN {X 0,Y 460.605,Z 1039.63,A -85,B 0,C 180,E1 20294.519,E2 20294.519} C_VEL
LIN {X 0,Y 453.291,Z 1058.55,A -85,B 0,C 180,E1 20292.049,E2 20292.049} C_VEL
LIN {X 0,Y 447.572,Z 1073.166,A -85,B 0,C 180,E1 20289.877,E2 20289.877} C_VEL
LIN {X 0,Y 442.29,Z 1086.661,A -85,B 0,C 180,E1 20287.616,E2 20287.616} C_VEL
LIN {X 0,Y 436.928,Z 1100.528,A -85,B 0,C 180,E1 20284.988,E2 20284.988} C_VEL
LIN {X 0,Y 430.919,Z 1116.474,A -85,B 0,C 180,E1 20281.471,E2 20281.471} C_VEL
LIN {X 0,Y 426.892,Z 1127.808,A -85,B 0,C 180,E1 20278.542,E2 20278.542} C_VEL
LIN {X 0,Y 423.769,Z 1137.321,A -85,B 0,C 180,E1 20275.73,E2 20275.73} C_VEL
LIN {X 0,Y 421.066,Z 1146.447,A -85,B 0,C 180,E1 20272.624,E2 20272.624} C_VEL
LIN {X 0,Y 418.608,Z 1156.127,A -85,B 0,C 180,E1 20268.667,E2 20268.667} C_VEL
LIN {X 0,Y 417.317,Z 1162.528,A -85,B 0,C 180,E1 20265.423,E2 20265.423} C_VEL
LIN {X 0,Y 416.582,Z 1167.274,A -85,B 0,C 180,E1 20262.475,E2 20262.475} C_VEL
LIN {X 0,Y 416.548,Z 1167.561,A -85,B 0,C 180,E1 20262.274,E2 20262.274} C_VEL
LIN {X 0,Y 415.39,Z 1169.132,A -85,B 0,C 180,E1 20261.237,E2 20261.237} C_VEL
LIN {X 0,Y 408.624,Z 1172.744,A -85,B 0,C 180,E1 20258.308,E2 20258.308} C_VEL
LIN {X 0,Y 408.056,Z 1173.367,A -85,B 0,C 180,E1 20257.535,E2 20257.535} C_VEL
LIN {X 0,Y 407.954,Z 1175.384,A -85,B 0,C 180,E1 20254.498,E2 20254.498} C_VEL
LIN {X 0,Y 407.933,Z 1176.357,A -85,B 0,C 180,E1 20251.685,E2 20251.685} C_VEL
LIN {X 0,Y 407.933,Z 1176.459,A -85,B 0,C 180,E1 20248.876,E2 20248.876} C_VEL
LIN {X 0,Y 407.951,Z 1175.659,A -85,B 0,C 180,E1 20246.001,E2 20246.001} C_VEL
LIN {X 0,Y 408.019,Z 1173.934,A -85,B 0,C 180,E1 20243.104,E2 20243.104} C_VEL
LIN {X 0,Y 408.21,Z 1171.356,A -85,B 0,C 180,E1 20240.27,E2 20240.27} C_VEL
LIN {X 0,Y 408.631,Z 1167.669,A -85,B 0,C 180,E1 20237.278,E2 20237.278} C_VEL
LIN {X 0,Y 409.361,Z 1163.199,A -85,B 0,C 180,E1 20234.415,E2 20234.415} C_VEL
LIN {X 0,Y 410.602,Z 1157.299,A -85,B 0,C 180,E1 20231.314,E2 20231.314} C_VEL
LIN {X 0,Y 412.841,Z 1148.907,A -85,B 0,C 180,E1 20227.652,E2 20227.652} C_VEL
LIN {X 0,Y 415.932,Z 1138.713,A -85,B 0,C 180,E1 20224.039,E2 20224.039} C_VEL
LIN {X 0,Y 419.31,Z 1128.881,A -85,B 0,C 180,E1 20221.049,E2 20221.049} C_VEL
LIN {X 0,Y 423.262,Z 1118.2,A -85,B 0,C 180,E1 20218.212,E2 20218.212} C_VEL
LIN {X 0,Y 428.763,Z 1104.298,A -85,B 0,C 180,E1 20214.994,E2 20214.994} C_VEL
LIN {X 0,Y 434.948,Z 1088.889,A -85,B 0,C 180,E1 20211.97,E2 20211.97} C_VEL
LIN {X 0,Y 440.701,Z 1074.748,A -85,B 0,C 180,E1 20209.543,E2 20209.543} C_VEL
LIN {X 0,Y 446.731,Z 1059.925,A -85,B 0,C 180,E1 20207.3,E2 20207.3} C_VEL
LIN {X 0,Y 453.315,Z 1043.479,A -85,B 0,C 180,E1 20205.105,E2 20205.105} C_VEL
LIN {X 0,Y 461.755,Z 1021.551,A -85,B 0,C 180,E1 20202.59,E2 20202.59} C_VEL
LIN {X 0,Y 468.581,Z 1002.877,A -85,B 0,C 180,E1 20200.756,E2 20200.756} C_VEL
LIN {X 0,Y 474.845,Z 984.853,A -85,B 0,C 180,E1 20199.206,E2 20199.206} C_VEL
LIN {X 0,Y 480.894,Z 966.312,A -85,B 0,C 180,E1 20197.807,E2 20197.807} C_VEL
LIN {X 0,Y 487.995,Z 942.77,A -85,B 0,C 180,E1 20196.27,E2 20196.27} C_VEL
LIN {X 0,Y 494.214,Z 919.131,A -85,B 0,C 180,E1 20194.979,E2 20194.979} C_VEL
LIN {X 0,Y 498.984,Z 899.07,A -85,B 0,C 180,E1 20194.049,E2 20194.049} C_VEL
LIN {X 0,Y 503.279,Z 878.6,A -85,B 0,C 180,E1 20193.239,E2 20193.239} C_VEL
LIN {X 0,Y 507.203,Z 856.928,A -85,B 0,C 180,E1 20192.523,E2 20192.523} C_VEL
LIN {X 0,Y 511.202,Z 830.08,A -85,B 0,C 180,E1 20191.813,E2 20191.813} C_VEL
LIN {X 0,Y 513.968,Z 803.599,A -85,B 0,C 180,E1 20191.301,E2 20191.301} C_VEL
LIN {X 0,Y 521.778,Z 678.845,A -85,B 0,C 180,E1 20189.352,E2 20189.352} C_VEL
LIN {X 0,Y 533.502,Z 494.074,A -85,B 0,C 180,E1 20186.476,E2 20186.476} C_VEL
LIN {X 0,Y 524.121,Z 480.228,A -85,B 0,C 180,E1 20183.856,E2 20183.856} C_VEL
LIN {X 0,Y 515.169,Z 467.491,A -85,B 0,C 180,E1 20180.983,E2 20180.983} C_VEL
LIN {X 0,Y 507.57,Z 457.258,A -85,B 0,C 180,E1 20178.135,E2 20178.135} C_VEL
LIN {X 0,Y 503.249,Z 451.73,A -85,B 0,C 180,E1 20176.269,E2 20176.269} C_VEL
LIN {X 0,Y 499.411,Z 446.708,A -85,B 0,C 180,E1 20174.375,E2 20174.375} C_VEL
LIN {X 0,Y 496.042,Z 442.398,A -85,B 0,C 180,E1 20172.456,E2 20172.456} C_VEL
LIN {X 0,Y 495.152,Z 441.179,A -85,B 0,C 180,E1 20171.887,E2 20171.887} C_VEL
LIN {X 0,Y 492.003,Z 437.651,A -85,B 0,C 180,E1 20169.652,E2 20169.652} C_VEL
LIN {X 0,Y 490.801,Z 435.454,A -85,B 0,C 180,E1 20168.553,E2 20168.553} C_VEL
LIN {X 0,Y 487.441,Z 432.09,A -85,B 0,C 180,E1 20164.589,E2 20164.589} C_VEL
LIN {X 0,Y 486.689,Z 429.408,A -85,B 0,C 180,E1 20162.355,E2 20162.355} C_VEL
LIN {X 0,Y 486.77,Z 429.577,A -85,B 0,C 180,E1 20157.763,E2 20157.763} C_VEL
LIN {X 0,Y 488.753,Z 433.968,A -85,B 0,C 180,E1 20153.893,E2 20153.893} C_VEL
LIN {X 0,Y 491.199,Z 435.879,A -85,B 0,C 180,E1 20151.513,E2 20151.513} C_VEL
LIN {X 0,Y 493.997,Z 440.23,A -85,B 0,C 180,E1 20149.268,E2 20149.268} C_VEL
LIN {X 0,Y 495.878,Z 442.051,A -85,B 0,C 180,E1 20148.072,E2 20148.072} C_VEL
LIN {X 0,Y 499.315,Z 446.541,A -85,B 0,C 180,E1 20146.096,E2 20146.096} C_VEL
LIN {X 0,Y 500.93,Z 448.783,A -85,B 0,C 180,E1 20145.256,E2 20145.256} C_VEL
LIN {X 0,Y 505.098,Z 454.142,A -85,B 0,C 180,E1 20143.319,E2 20143.319} C_VEL
LIN {X 0,Y 510.913,Z 462.832,A -85,B 0,C 180,E1 20140.923,E2 20140.923} C_VEL
LIN {X 0,Y 516.763,Z 471.642,A -85,B 0,C 180,E1 20138.817,E2 20138.817} C_VEL
LIN {X 0,Y 524.94,Z 484.593,A -85,B 0,C 180,E1 20136.213,E2 20136.213} C_VEL
LIN {X 0,Y 533.583,Z 499.062,A -85,B 0,C 180,E1 20133.775,E2 20133.775} C_VEL
LIN {X 0,Y 520.037,Z 714.415,A -85,B 0,C 180,E1 20130.428,E2 20130.428} C_VEL
LIN {X 0,Y 513.386,Z 821.432,A -85,B 0,C 180,E1 20128.751,E2 20128.751} C_VEL
LIN {X 0,Y 510.414,Z 849.109,A -85,B 0,C 180,E1 20128.223,E2 20128.223} C_VEL
LIN {X 0,Y 506.315,Z 875.38,A -85,B 0,C 180,E1 20127.555,E2 20127.555} C_VEL
LIN {X 0,Y 502.353,Z 896.771,A -85,B 0,C 180,E1 20126.87,E2 20126.87} C_VEL
LIN {X 0,Y 498.049,Z 916.929,A -85,B 0,C 180,E1 20126.101,E2 20126.101} C_VEL
LIN {X 0,Y 493.211,Z 937.176,A -85,B 0,C 180,E1 20125.188,E2 20125.188} C_VEL
LIN {X 0,Y 486.826,Z 961.309,A -85,B 0,C 180,E1 20123.908,E2 20123.908} C_VEL
LIN {X 0,Y 479.65,Z 985.227,A -85,B 0,C 180,E1 20122.385,E2 20122.385} C_VEL
LIN {X 0,Y 473.308,Z 1004.891,A -85,B 0,C 180,E1 20120.926,E2 20120.926} C_VEL
LIN {X 0,Y 466.801,Z 1023.927,A -85,B 0,C 180,E1 20119.309,E2 20119.309} C_VEL
LIN {X 0,Y 459.009,Z 1045.707,A -85,B 0,C 180,E1 20117.183,E2 20117.183} C_VEL
LIN {X 0,Y 451.178,Z 1066.302,A -85,B 0,C 180,E1 20114.807,E2 20114.807} C_VEL
LIN {X 0,Y 445.057,Z 1082.138,A -85,B 0,C 180,E1 20112.721,E2 20112.721} C_VEL
LIN {X 0,Y 439.144,Z 1097.349,A -85,B 0,C 180,E1 20110.458,E2 20110.458} C_VEL
LIN {X 0,Y 432.542,Z 1114.573,A -85,B 0,C 180,E1 20107.542,E2 20107.542} C_VEL
LIN {X 0,Y 426.432,Z 1130.509,A -85,B 0,C 180,E1 20104.374,E2 20104.374} C_VEL
LIN {X 0,Y 421.979,Z 1142.796,A -85,B 0,C 180,E1 20101.577,E2 20101.577} C_VEL
LIN {X 0,Y 418.237,Z 1153.848,A -85,B 0,C 180,E1 20098.719,E2 20098.719} C_VEL
LIN {X 0,Y 414.526,Z 1165.969,A -85,B 0,C 180,E1 20095.12,E2 20095.12} C_VEL
LIN {X 0,Y 411.799,Z 1176.03,A -85,B 0,C 180,E1 20091.508,E2 20091.508} C_VEL
LIN {X 0,Y 410.177,Z 1183.22,A -85,B 0,C 180,E1 20088.475,E2 20088.475} C_VEL
LIN {X 0,Y 409.108,Z 1189.261,A -85,B 0,C 180,E1 20085.45,E2 20085.45} C_VEL
LIN {X 0,Y 408.458,Z 1193.98,A -85,B 0,C 180,E1 20082.583,E2 20082.583} C_VEL
LIN {X 0,Y 408.112,Z 1197.88,A -85,B 0,C 180,E1 20079.59,E2 20079.59} C_VEL
LIN {X 0,Y 407.971,Z 1200.723,A -85,B 0,C 180,E1 20076.614,E2 20076.614} C_VEL
LIN {X 0,Y 407.933,Z 1202.595,A -85,B 0,C 180,E1 20073.513,E2 20073.513} C_VEL
LIN {X 0,Y 407.937,Z 1203.403,A -85,B 0,C 180,E1 20070,E2 20070} C_VEL
LIN {X 0,Y 407.933,Z 1202.594,A -85,B 0,C 180,E1 20066.487,E2 20066.487} C_VEL
LIN {X 0,Y 407.971,Z 1200.722,A -85,B 0,C 180,E1 20063.386,E2 20063.386} C_VEL
LIN {X 0,Y 408.112,Z 1197.88,A -85,B 0,C 180,E1 20060.41,E2 20060.41} C_VEL
LIN {X 0,Y 408.458,Z 1193.98,A -85,B 0,C 180,E1 20057.417,E2 20057.417} C_VEL
LIN {X 0,Y 409.108,Z 1189.261,A -85,B 0,C 180,E1 20054.55,E2 20054.55} C_VEL
LIN {X 0,Y 410.177,Z 1183.217,A -85,B 0,C 180,E1 20051.525,E2 20051.525} C_VEL
LIN {X 0,Y 411.892,Z 1175.663,A -85,B 0,C 180,E1 20048.348,E2 20048.348} C_VEL
LIN {X 0,Y 414.912,Z 1164.564,A -85,B 0,C 180,E1 20044.447,E2 20044.447} C_VEL
LIN {X 0,Y 418.239,Z 1153.847,A -85,B 0,C 180,E1 20041.281,E2 20041.281} C_VEL
LIN {X 0,Y 421.979,Z 1142.791,A -85,B 0,C 180,E1 20038.423,E2 20038.423} C_VEL
LIN {X 0,Y 426.429,Z 1130.5,A -85,B 0,C 180,E1 20035.626,E2 20035.626} C_VEL
LIN {X 0,Y 432.648,Z 1114.24,A -85,B 0,C 180,E1 20032.403,E2 20032.403} C_VEL
LIN {X 0,Y 439.139,Z 1097.318,A -85,B 0,C 180,E1 20029.541,E2 20029.541} C_VEL
LIN {X 0,Y 445.056,Z 1082.087,A -85,B 0,C 180,E1 20027.276,E2 20027.276} C_VEL
LIN {X 0,Y 451.285,Z 1065.957,A -85,B 0,C 180,E1 20025.155,E2 20025.155} C_VEL
LIN {X 0,Y 459.327,Z 1044.718,A -85,B 0,C 180,E1 20022.721,E2 20022.721} C_VEL
LIN {X 0,Y 466.79,Z 1023.842,A -85,B 0,C 180,E1 20020.689,E2 20020.689} C_VEL
LIN {X 0,Y 473.296,Z 1004.79,A -85,B 0,C 180,E1 20019.072,E2 20019.072} C_VEL
LIN {X 0,Y 479.897,Z 984.297,A -85,B 0,C 180,E1 20017.556,E2 20017.556} C_VEL
LIN {X 0,Y 487.702,Z 957.791,A -85,B 0,C 180,E1 20015.899,E2 20015.899} C_VEL
LIN {X 0,Y 493.195,Z 937.013,A -85,B 0,C 180,E1 20014.809,E2 20014.809} C_VEL
LIN {X 0,Y 498.141,Z 916.256,A -85,B 0,C 180,E1 20013.877,E2 20013.877} C_VEL
LIN {X 0,Y 502.487,Z 895.794,A -85,B 0,C 180,E1 20013.101,E2 20013.101} C_VEL
LIN {X 0,Y 506.606,Z 873.36,A -85,B 0,C 180,E1 20012.392,E2 20012.392} C_VEL
LIN {X 0,Y 510.921,Z 844.26,A -85,B 0,C 180,E1 20011.682,E2 20011.682} C_VEL
LIN {X 0,Y 513.424,Z 820.032,A -85,B 0,C 180,E1 20011.231,E2 20011.231} C_VEL
LIN {X 0,Y 526.266,Z 612.208,A -85,B 0,C 180,E1 20007.99,E2 20007.99} C_VEL
LIN {X 0,Y 533.474,Z 498.913,A -85,B 0,C 180,E1 20006.223,E2 20006.223} C_VEL
LIN {X 0,Y 523.982,Z 483.081,A -85,B 0,C 180,E1 20003.535,E2 20003.535} C_VEL
LIN {X 0,Y 515.264,Z 469.356,A -85,B 0,C 180,E1 20000.712,E2 20000.712} C_VEL
LIN {X 0,Y 508.301,Z 459.009,A -85,B 0,C 180,E1 19998.108,E2 19998.108} C_VEL
LIN {X 0,Y 503.593,Z 452.124,A -85,B 0,C 180,E1 19996.08,E2 19996.08} C_VEL
LIN {X 0,Y 499.252,Z 446.522,A -85,B 0,C 180,E1 19993.965,E2 19993.965} C_VEL
LIN {X 0,Y 495.703,Z 441.825,A -85,B 0,C 180,E1 19991.932,E2 19991.932} C_VEL
LIN {X 0,Y 492.032,Z 437.682,A -85,B 0,C 180,E1 19989.415,E2 19989.415} C_VEL
LIN {X 0,Y 490.795,Z 435.468,A -85,B 0,C 180,E1 19988.317,E2 19988.317} C_VEL
LIN {X 0,Y 487.458,Z 432.18,A -85,B 0,C 180,E1 19984.588,E2 19984.588} C_VEL
LIN {X 0,Y 486.565,Z 429.395,A -85,B 0,C 180,E1 19982.356,E2 19982.356} C_VEL
LIN {X 0,Y 486.671,Z 429.6,A -85,B 0,C 180,E1 19976.82,E2 19976.82} C_VEL
LIN {X 0,Y 487.808,Z 432.755,A -85,B 0,C 180,E1 19974.354,E2 19974.354} C_VEL
LIN {X 0,Y 491.071,Z 435.859,A -85,B 0,C 180,E1 19970.929,E2 19970.929} C_VEL
LIN {X 0,Y 493.592,Z 439.819,A -85,B 0,C 180,E1 19968.904,E2 19968.904} C_VEL
LIN {X 0,Y 495.734,Z 441.946,A -85,B 0,C 180,E1 19967.536,E2 19967.536} C_VEL
LIN {X 0,Y 499.072,Z 446.424,A -85,B 0,C 180,E1 19965.615,E2 19965.615} C_VEL
LIN {X 0,Y 500.595,Z 448.386,A -85,B 0,C 180,E1 19964.831,E2 19964.831} C_VEL
LIN {X 0,Y 504.759,Z 453.69,A -85,B 0,C 180,E1 19962.892,E2 19962.892} C_VEL
LIN {X 0,Y 509.109,Z 459.524,A -85,B 0,C 180,E1 19961.091,E2 19961.091} C_VEL
LIN {X 0,Y 515.348,Z 467.823,A -85,B 0,C 180,E1 19958.816,E2 19958.816} C_VEL
LIN {X 0,Y 525.329,Z 481.96,A -85,B 0,C 180,E1 19955.664,E2 19955.664} C_VEL
LIN {X 0,Y 533.433,Z 494.159,A -85,B 0,C 180,E1 19953.42,E2 19953.42} C_VEL
LIN {X 0,Y 519.816,Z 709.33,A -85,B 0,C 180,E1 19950.082,E2 19950.082} C_VEL
LIN {X 0,Y 513.852,Z 804.131,A -85,B 0,C 180,E1 19948.595,E2 19948.595} C_VEL
LIN {X 0,Y 510.932,Z 831.632,A -85,B 0,C 180,E1 19948.057,E2 19948.057} C_VEL
LIN {X 0,Y 507.044,Z 857.451,A -85,B 0,C 180,E1 19947.366,E2 19947.366} C_VEL
LIN {X 0,Y 503.219,Z 878.555,A -85,B 0,C 180,E1 19946.668,E2 19946.668} C_VEL
LIN {X 0,Y 498.932,Z 899.022,A -85,B 0,C 180,E1 19945.858,E2 19945.858} C_VEL
LIN {X 0,Y 493.622,Z 921.33,A -85,B 0,C 180,E1 19944.816,E2 19944.816} C_VEL
LIN {X 0,Y 486.322,Z 948.132,A -85,B 0,C 180,E1 19943.304,E2 19943.304} C_VEL
LIN {X 0,Y 480.322,Z 967.93,A -85,B 0,C 180,E1 19941.981,E2 19941.981} C_VEL
LIN {X 0,Y 474.549,Z 985.584,A -85,B 0,C 180,E1 19940.638,E2 19940.638} C_VEL
LIN {X 0,Y 468.324,Z 1003.471,A -85,B 0,C 180,E1 19939.093,E2 19939.093} C_VEL
LIN {X 0,Y 461.095,Z 1023.291,A -85,B 0,C 180,E1 19937.133,E2 19937.133} C_VEL
LIN {X 0,Y 452.984,Z 1044.234,A -85,B 0,C 180,E1 19934.703,E2 19934.703} C_VEL
LIN {X 0,Y 446.911,Z 1059.412,A -85,B 0,C 180,E1 19932.679,E2 19932.679} C_VEL
LIN {X 0,Y 441.209,Z 1073.442,A -85,B 0,C 180,E1 19930.571,E2 19930.571} C_VEL
LIN {X 0,Y 435.406,Z 1087.694,A -85,B 0,C 180,E1 19928.15,E2 19928.15} C_VEL
LIN {X 0,Y 429.175,Z 1103.262,A -85,B 0,C 180,E1 19925.13,E2 19925.13} C_VEL
LIN {X 0,Y 423.355,Z 1117.945,A -85,B 0,C 180,E1 19921.76,E2 19921.76} C_VEL
LIN {X 0,Y 419.413,Z 1128.586,A -85,B 0,C 180,E1 19918.943,E2 19918.943} C_VEL
LIN {X 0,Y 416.15,Z 1138.043,A -85,B 0,C 180,E1 19916.084,E2 19916.084} C_VEL
LIN {X 0,Y 413.008,Z 1148.299,A -85,B 0,C 180,E1 19912.489,E2 19912.489} C_VEL
LIN {X 0,Y 410.653,Z 1157.068,A -85,B 0,C 180,E1 19908.707,E2 19908.707} C_VEL
LIN {X 0,Y 409.392,Z 1163.044,A -85,B 0,C 180,E1 19905.584,E2 19905.584} C_VEL
LIN {X 0,Y 408.644,Z 1167.542,A -85,B 0,C 180,E1 19902.721,E2 19902.721} C_VEL
LIN {X 0,Y 408.22,Z 1171.256,A -85,B 0,C 180,E1 19899.73,E2 19899.73} C_VEL
LIN {X 0,Y 408.056,Z 1173.367,A -85,B 0,C 180,E1 19897.535,E2 19897.535} C_VEL
LIN {X 0,Y 407.032,Z 1174.25,A -85,B 0,C 180,E1 19896.461,E2 19896.461} C_VEL
LIN {X 0,Y 402.35,Z 1175.768,A -85,B 0,C 180,E1 19894.434,E2 19894.434} C_VEL
LIN {X 0,Y 400.091,Z 1176.399,A -85,B 0,C 180,E1 19893.033,E2 19893.033} C_VEL
LIN {X 0,Y 399.942,Z 1176.483,A -85,B 0,C 180,E1 19892.633,E2 19892.633} C_VEL
LIN {X 0,Y 399.933,Z 1176.765,A -85,B 0,C 180,E1 19889.141,E2 19889.141} C_VEL
LIN {X 0,Y 399.955,Z 1176.018,A -85,B 0,C 180,E1 19886.13,E2 19886.13} C_VEL
LIN {X 0,Y 400.028,Z 1174.307,A -85,B 0,C 180,E1 19883.109,E2 19883.109} C_VEL
LIN {X 0,Y 400.227,Z 1171.775,A -85,B 0,C 180,E1 19880.219,E2 19880.219} C_VEL
LIN {X 0,Y 400.669,Z 1168.135,A -85,B 0,C 180,E1 19877.168,E2 19877.168} C_VEL
LIN {X 0,Y 401.438,Z 1163.713,A -85,B 0,C 180,E1 19874.247,E2 19874.247} C_VEL
LIN {X 0,Y 402.698,Z 1158.029,A -85,B 0,C 180,E1 19871.169,E2 19871.169} C_VEL
LIN {X 0,Y 404.647,Z 1150.895,A -85,B 0,C 180,E1 19867.94,E2 19867.94} C_VEL
LIN {X 0,Y 408.016,Z 1140.375,A -85,B 0,C 180,E1 19863.983,E2 19863.983} C_VEL
LIN {X 0,Y 411.851,Z 1129.656,A -85,B 0,C 180,E1 19860.633,E2 19860.633} C_VEL
LIN {X 0,Y 415.957,Z 1119.033,A -85,B 0,C 180,E1 19857.749,E2 19857.749} C_VEL
LIN {X 0,Y 420.855,Z 1107.061,A -85,B 0,C 180,E1 19854.905,E2 19854.905} C_VEL
LIN {X 0,Y 428.093,Z 1089.917,A -85,B 0,C 180,E1 19851.42,E2 19851.42} C_VEL
LIN {X 0,Y 434.393,Z 1075.019,A -85,B 0,C 180,E1 19848.83,E2 19848.83} C_VEL
LIN {X 0,Y 440.663,Z 1060.16,A -85,B 0,C 180,E1 19846.561,E2 19846.561} C_VEL
LIN {X 0,Y 447.658,Z 1043.306,A -85,B 0,C 180,E1 19844.298,E2 19844.298} C_VEL
LIN {X 0,Y 456.21,Z 1021.818,A -85,B 0,C 180,E1 19841.827,E2 19841.827} C_VEL
LIN {X 0,Y 463.252,Z 1003.142,A -85,B 0,C 180,E1 19839.985,E2 19839.985} C_VEL
LIN {X 0,Y 469.874,Z 984.627,A -85,B 0,C 180,E1 19838.391,E2 19838.391} C_VEL
LIN {X 0,Y 476.699,Z 964.24,A -85,B 0,C 180,E1 19836.863,E2 19836.863} C_VEL
LIN {X 0,Y 484.31,Z 939.041,A -85,B 0,C 180,E1 19835.263,E2 19835.263} C_VEL
LIN {X 0,Y 489.918,Z 918.19,A -85,B 0,C 180,E1 19834.143,E2 19834.143} C_VEL
LIN {X 0,Y 494.801,Z 898.049,A -85,B 0,C 180,E1 19833.22,E2 19833.22} C_VEL
LIN {X 0,Y 499.205,Z 877.382,A -85,B 0,C 180,E1 19832.412,E2 19832.412} C_VEL
LIN {X 0,Y 503.772,Z 852.452,A -85,B 0,C 180,E1 19831.61,E2 19831.61} C_VEL
LIN {X 0,Y 507.614,Z 825.168,A -85,B 0,C 180,E1 19830.936,E2 19830.936} C_VEL
LIN {X 0,Y 509.979,Z 802.302,A -85,B 0,C 180,E1 19830.506,E2 19830.506} C_VEL
LIN {X 0,Y 523.46,Z 592.977,A -85,B 0,C 180,E1 19827.242,E2 19827.242} C_VEL
LIN {X 0,Y 529.629,Z 498.883,A -85,B 0,C 180,E1 19825.763,E2 19825.763} C_VEL
LIN {X 0,Y 520.163,Z 484.736,A -85,B 0,C 180,E1 19822.998,E2 19822.998} C_VEL
LIN {X 0,Y 512.055,Z 473.333,A -85,B 0,C 180,E1 19820.28,E2 19820.28} C_VEL
LIN {X 0,Y 505.79,Z 464.654,A -85,B 0,C 180,E1 19817.844,E2 19817.844} C_VEL
LIN {X 0,Y 501.671,Z 459.29,A -85,B 0,C 180,E1 19816.025,E2 19816.025} C_VEL
LIN {X 0,Y 498.009,Z 454.41,A -85,B 0,C 180,E1 19814.179,E2 19814.179} C_VEL
LIN {X 0,Y 494.698,Z 450.098,A -85,B 0,C 180,E1 19812.253,E2 19812.253} C_VEL
LIN {X 0,Y 493.64,Z 448.772,A -85,B 0,C 180,E1 19811.568,E2 19811.568} C_VEL
LIN {X 0,Y 490.617,Z 445.102,A -85,B 0,C 180,E1 19809.324,E2 19809.324} C_VEL
LIN {X 0,Y 489.699,Z 443.342,A -85,B 0,C 180,E1 19808.454,E2 19808.454} C_VEL
LIN {X 0,Y 486.402,Z 439.969,A -85,B 0,C 180,E1 19804.48,E2 19804.48} C_VEL
LIN {X 0,Y 485.678,Z 437.346,A -85,B 0,C 180,E1 19802.242,E2 19802.242} C_VEL
LIN {X 0,Y 485.76,Z 437.466,A -85,B 0,C 180,E1 19797.877,E2 19797.877} C_VEL
LIN {X 0,Y 487.682,Z 441.849,A -85,B 0,C 180,E1 19793.998,E2 19793.998} C_VEL
LIN {X 0,Y 490.081,Z 443.842,A -85,B 0,C 180,E1 19791.612,E2 19791.612} C_VEL
LIN {X 0,Y 492.857,Z 448.114,A -85,B 0,C 180,E1 19789.361,E2 19789.361} C_VEL
LIN {X 0,Y 494.621,Z 449.904,A -85,B 0,C 180,E1 19788.219,E2 19788.219} C_VEL
LIN {X 0,Y 498.13,Z 454.44,A -85,B 0,C 180,E1 19786.18,E2 19786.18} C_VEL
LIN {X 0,Y 503.61,Z 461.871,A -85,B 0,C 180,E1 19783.506,E2 19783.506} C_VEL
LIN {X 0,Y 509.352,Z 470.617,A -85,B 0,C 180,E1 19781.101,E2 19781.101} C_VEL
LIN {X 0,Y 516.068,Z 480.915,A -85,B 0,C 180,E1 19778.668,E2 19778.668} C_VEL
LIN {X 0,Y 524.602,Z 494.884,A -85,B 0,C 180,E1 19775.958,E2 19775.958} C_VEL
LIN {X 0,Y 529.732,Z 503.863,A -85,B 0,C 180,E1 19774.478,E2 19774.478} C_VEL
LIN {X 0,Y 515.667,Z 721.191,A -85,B 0,C 180,E1 19771.097,E2 19771.097} C_VEL
LIN {X 0,Y 509.247,Z 821.295,A -85,B 0,C 180,E1 19769.524,E2 19769.524} C_VEL
LIN {X 0,Y 506.186,Z 849.057,A -85,B 0,C 180,E1 19768.994,E2 19768.994} C_VEL
LIN {X 0,Y 502.004,Z 875.234,A -85,B 0,C 180,E1 19768.33,E2 19768.33} C_VEL
LIN {X 0,Y 497.967,Z 896.513,A -85,B 0,C 180,E1 19767.652,E2 19767.652} C_VEL
LIN {X 0,Y 493.586,Z 916.54,A -85,B 0,C 180,E1 19766.89,E2 19766.89} C_VEL
LIN {X 0,Y 488.59,Z 936.914,A -85,B 0,C 180,E1 19765.975,E2 19765.975} C_VEL
LIN {X 0,Y 482.057,Z 960.944,A -85,B 0,C 180,E1 19764.704,E2 19764.704} C_VEL
LIN {X 0,Y 474.652,Z 984.961,A -85,B 0,C 180,E1 19763.175,E2 19763.175} C_VEL
LIN {X 0,Y 468.219,Z 1004.362,A -85,B 0,C 180,E1 19761.735,E2 19761.735} C_VEL
LIN {X 0,Y 461.91,Z 1022.308,A -85,B 0,C 180,E1 19760.214,E2 19760.214} C_VEL
LIN {X 0,Y 455.3,Z 1040.206,A -85,B 0,C 180,E1 19758.491,E2 19758.491} C_VEL
LIN {X 0,Y 447.38,Z 1060.89,A -85,B 0,C 180,E1 19756.21,E2 19756.21} C_VEL
LIN {X 0,Y 439.423,Z 1080.59,A -85,B 0,C 180,E1 19753.647,E2 19753.647} C_VEL
LIN {X 0,Y 433.348,Z 1095.592,A -85,B 0,C 180,E1 19751.419,E2 19751.419} C_VEL
LIN {X 0,Y 427.485,Z 1110.069,A -85,B 0,C 180,E1 19748.989,E2 19748.989} C_VEL
LIN {X 0,Y 421.136,Z 1126.186,A -85,B 0,C 180,E1 19745.904,E2 19745.904} C_VEL
LIN {X 0,Y 415.454,Z 1140.809,A -85,B 0,C 180,E1 19742.609,E2 19742.609} C_VEL
LIN {X 0,Y 411.402,Z 1151.993,A -85,B 0,C 180,E1 19739.722,E2 19739.722} C_VEL
LIN {X 0,Y 408.079,Z 1161.943,A -85,B 0,C 180,E1 19736.797,E2 19736.797} C_VEL
LIN {X 0,Y 405.329,Z 1171.105,A -85,B 0,C 180,E1 19733.709,E2 19733.709} C_VEL
LIN {X 0,Y 402.787,Z 1181.078,A -85,B 0,C 180,E1 19729.731,E2 19729.731} C_VEL
LIN {X 0,Y 401.326,Z 1188.206,A -85,B 0,C 180,E1 19726.203,E2 19726.203} C_VEL
LIN {X 0,Y 400.551,Z 1193.286,A -85,B 0,C 180,E1 19723.13,E2 19723.13} C_VEL
LIN {X 0,Y 400.167,Z 1197.12,A -85,B 0,C 180,E1 19720.218,E2 19720.218} C_VEL
LIN {X 0,Y 400.001,Z 1199.989,A -85,B 0,C 180,E1 19717.324,E2 19717.324} C_VEL
LIN {X 0,Y 399.939,Z 1201.91,A -85,B 0,C 180,E1 19714.445,E2 19714.445} C_VEL
LIN {X 0,Y 399.938,Z 1202.869,A -85,B 0,C 180,E1 19711.719,E2 19711.719} C_VEL
LIN {X 0,Y 399.94,Z 1202.963,A -85,B 0,C 180,E1 19708.854,E2 19708.854} C_VEL
LIN {X 0,Y 399.937,Z 1202.121,A -85,B 0,C 180,E1 19705.986,E2 19705.986} C_VEL
LIN {X 0,Y 399.977,Z 1200.34,A -85,B 0,C 180,E1 19703.109,E2 19703.109} C_VEL
LIN {X 0,Y 400.129,Z 1197.613,A -85,B 0,C 180,E1 19700.217,E2 19700.217} C_VEL
LIN {X 0,Y 400.497,Z 1193.712,A -85,B 0,C 180,E1 19697.162,E2 19697.162} C_VEL
LIN {X 0,Y 401.198,Z 1188.991,A -85,B 0,C 180,E1 19694.238,E2 19694.238} C_VEL
LIN {X 0,Y 402.34,Z 1182.945,A -85,B 0,C 180,E1 19691.152,E2 19691.152} C_VEL
LIN {X 0,Y 404.163,Z 1175.389,A -85,B 0,C 180,E1 19687.912,E2 19687.912} C_VEL
LIN {X 0,Y 407.359,Z 1164.287,A -85,B 0,C 180,E1 19683.937,E2 19683.937} C_VEL
LIN {X 0,Y 410.872,Z 1153.569,A -85,B 0,C 180,E1 19680.716,E2 19680.716} C_VEL
LIN {X 0,Y 414.588,Z 1143.098,A -85,B 0,C 180,E1 19677.956,E2 19677.956} C_VEL
LIN {X 0,Y 419.022,Z 1131.382,A -85,B 0,C 180,E1 19675.229,E2 19675.229} C_VEL
LIN {X 0,Y 424.491,Z 1117.602,A -85,B 0,C 180,E1 19672.407,E2 19672.407} C_VEL
LIN {X 0,Y 432.064,Z 1098.756,A -85,B 0,C 180,E1 19669.088,E2 19669.088} C_VEL
LIN {X 0,Y 438.501,Z 1082.797,A -85,B 0,C 180,E1 19666.669,E2 19666.669} C_VEL
LIN {X 0,Y 444.83,Z 1067.005,A -85,B 0,C 180,E1 19664.559,E2 19664.559} C_VEL
LIN {X 0,Y 452.111,Z 1048.478,A -85,B 0,C 180,E1 19662.383,E2 19662.383} C_VEL
LIN {X 0,Y 460.692,Z 1025.557,A -85,B 0,C 180,E1 19660.085,E2 19660.085} C_VEL
LIN {X 0,Y 467.602,Z 1005.998,A -85,B 0,C 180,E1 19658.402,E2 19658.402} C_VEL
LIN {X 0,Y 474.104,Z 986.477,A -85,B 0,C 180,E1 19656.938,E2 19656.938} C_VEL
LIN {X 0,Y 481.207,Z 963.633,A -85,B 0,C 180,E1 19655.462,E2 19655.462} C_VEL
LIN {X 0,Y 488.286,Z 937.876,A -85,B 0,C 180,E1 19654.077,E2 19654.077} C_VEL
LIN {X 0,Y 493.272,Z 917.62,A -85,B 0,C 180,E1 19653.16,E2 19653.16} C_VEL
LIN {X 0,Y 497.797,Z 897.006,A -85,B 0,C 180,E1 19652.371,E2 19652.371} C_VEL
LIN {X 0,Y 501.83,Z 875.807,A -85,B 0,C 180,E1 19651.692,E2 19651.692} C_VEL
LIN {X 0,Y 505.717,Z 851.616,A -85,B 0,C 180,E1 19651.071,E2 19651.071} C_VEL
LIN {X 0,Y 509.073,Z 822.493,A -85,B 0,C 180,E1 19650.502,E2 19650.502} C_VEL
LIN {X 0,Y 513.622,Z 752.66,A -85,B 0,C 180,E1 19649.398,E2 19649.398} C_VEL
LIN {X 0,Y 527.757,Z 532.147,A -85,B 0,C 180,E1 19645.969,E2 19645.969} C_VEL
LIN {X 0,Y 529.558,Z 503.491,A -85,B 0,C 180,E1 19645.499,E2 19645.499} C_VEL
LIN {X 0,Y 521.434,Z 489.719,A -85,B 0,C 180,E1 19643.118,E2 19643.118} C_VEL
LIN {X 0,Y 513.199,Z 476.503,A -85,B 0,C 180,E1 19640.381,E2 19640.381} C_VEL
LIN {X 0,Y 506.371,Z 466.18,A -85,B 0,C 180,E1 19637.763,E2 19637.763} C_VEL
LIN {X 0,Y 502.003,Z 459.687,A -85,B 0,C 180,E1 19635.836,E2 19635.836} C_VEL
LIN {X 0,Y 497.738,Z 454.113,A -85,B 0,C 180,E1 19633.712,E2 19633.712} C_VEL
LIN {X 0,Y 493.904,Z 449.042,A -85,B 0,C 180,E1 19631.443,E2 19631.443} C_VEL
LIN {X 0,Y 490.836,Z 445.491,A -85,B 0,C 180,E1 19629.261,E2 19629.261} C_VEL
LIN {X 0,Y 489.688,Z 443.358,A -85,B 0,C 180,E1 19628.218,E2 19628.218} C_VEL
LIN {X 0,Y 486.386,Z 440.003,A -85,B 0,C 180,E1 19624.436,E2 19624.436} C_VEL
LIN {X 0,Y 485.547,Z 437.328,A -85,B 0,C 180,E1 19622.242,E2 19622.242} C_VEL
LIN {X 0,Y 485.652,Z 437.497,A -85,B 0,C 180,E1 19616.931,E2 19616.931} C_VEL
LIN {X 0,Y 486.831,Z 440.748,A -85,B 0,C 180,E1 19614.342,E2 19614.342} C_VEL
LIN {X 0,Y 489.901,Z 443.712,A -85,B 0,C 180,E1 19611.076,E2 19611.076} C_VEL
LIN {X 0,Y 492.454,Z 447.706,A -85,B 0,C 180,E1 19608.997,E2 19608.997} C_VEL
LIN {X 0,Y 494.39,Z 449.651,A -85,B 0,C 180,E1 19607.739,E2 19607.739} C_VEL
LIN {X 0,Y 497.78,Z 454.225,A -85,B 0,C 180,E1 19605.755,E2 19605.755} C_VEL
LIN {X 0,Y 499.825,Z 457.065,A -85,B 0,C 180,E1 19604.689,E2 19604.689} C_VEL
LIN {X 0,Y 503.153,Z 461.241,A -85,B 0,C 180,E1 19603.134,E2 19603.134} C_VEL
LIN {X 0,Y 507.571,Z 467.277,A -85,B 0,C 180,E1 19601.27,E2 19601.27} C_VEL
LIN {X 0,Y 513.512,Z 475.323,A -85,B 0,C 180,E1 19599.065,E2 19599.065} C_VEL
LIN {X 0,Y 523.108,Z 489.116,A -85,B 0,C 180,E1 19595.975,E2 19595.975} C_VEL
LIN {X 0,Y 529.58,Z 499.122,A -85,B 0,C 180,E1 19594.123,E2 19594.123} C_VEL
LIN {X 0,Y 515.558,Z 714.566,A -85,B 0,C 180,E1 19590.775,E2 19590.775} C_VEL
LIN {X 0,Y 509.718,Z 804.524,A -85,B 0,C 180,E1 19589.361,E2 19589.361} C_VEL
LIN {X 0,Y 506.699,Z 832.169,A -85,B 0,C 180,E1 19588.819,E2 19588.819} C_VEL
LIN {X 0,Y 502.76,Z 857.726,A -85,B 0,C 180,E1 19588.137,E2 19588.137} C_VEL
LIN {X 0,Y 498.84,Z 878.83,A -85,B 0,C 180,E1 19587.441,E2 19587.441} C_VEL
LIN {X 0,Y 494.425,Z 899.395,A -85,B 0,C 180,E1 19586.628,E2 19586.628} C_VEL
LIN {X 0,Y 489.001,Z 921.603,A -85,B 0,C 180,E1 19585.592,E2 19585.592} C_VEL
LIN {X 0,Y 481.788,Z 947.513,A -85,B 0,C 180,E1 19584.135,E2 19584.135} C_VEL
LIN {X 0,Y 475.625,Z 967.33,A -85,B 0,C 180,E1 19582.819,E2 19582.819} C_VEL
LIN {X 0,Y 469.416,Z 985.788,A -85,B 0,C 180,E1 19581.417,E2 19581.417} C_VEL
LIN {X 0,Y 462.98,Z 1003.746,A -85,B 0,C 180,E1 19579.863,E2 19579.863} C_VEL
LIN {X 0,Y 455.517,Z 1023.566,A -85,B 0,C 180,E1 19577.894,E2 19577.894} C_VEL
LIN {X 0,Y 447.254,Z 1044.198,A -85,B 0,C 180,E1 19575.491,E2 19575.491} C_VEL
LIN {X 0,Y 440.641,Z 1060.144,A -85,B 0,C 180,E1 19573.346,E2 19573.346} C_VEL
LIN {X 0,Y 434.565,Z 1074.55,A -85,B 0,C 180,E1 19571.15,E2 19571.15} C_VEL
LIN {X 0,Y 428.252,Z 1089.485,A -85,B 0,C 180,E1 19568.563,E2 19568.563} C_VEL
LIN {X 0,Y 421.001,Z 1106.703,A -85,B 0,C 180,E1 19565.081,E2 19565.081} C_VEL
LIN {X 0,Y 416.058,Z 1118.765,A -85,B 0,C 180,E1 19562.226,E2 19562.226} C_VEL
LIN {X 0,Y 411.957,Z 1129.365,A -85,B 0,C 180,E1 19559.358,E2 19559.358} C_VEL
LIN {X 0,Y 408.397,Z 1139.213,A -85,B 0,C 180,E1 19556.304,E2 19556.304} C_VEL
LIN {X 0,Y 404.926,Z 1149.996,A -85,B 0,C 180,E1 19552.35,E2 19552.35} C_VEL
LIN {X 0,Y 402.804,Z 1157.593,A -85,B 0,C 180,E1 19548.955,E2 19548.955} C_VEL
LIN {X 0,Y 401.522,Z 1163.313,A -85,B 0,C 180,E1 19545.898,E2 19545.898} C_VEL
LIN {X 0,Y 400.711,Z 1167.81,A -85,B 0,C 180,E1 19542.977,E2 19542.977} C_VEL
LIN {X 0,Y 400.25,Z 1171.522,A -85,B 0,C 180,E1 19539.925,E2 19539.925} C_VEL
LIN {X 0,Y 400.038,Z 1174.127,A -85,B 0,C 180,E1 19537.035,E2 19537.035} C_VEL
LIN {X 0,Y 399.957,Z 1175.844,A -85,B 0,C 180,E1 19534.157,E2 19534.157} C_VEL
LIN {X 0,Y 399.942,Z 1176.483,A -85,B 0,C 180,E1 19532.633,E2 19532.633} C_VEL
LIN {X 0,Y 398.94,Z 1176.718,A -85,B 0,C 180,E1 19531.53,E2 19531.53} C_VEL
LIN {X 0,Y 394.145,Z 1177.01,A -85,B 0,C 180,E1 19529.37,E2 19529.37} C_VEL
LIN {X 0,Y 392.088,Z 1176.862,A -85,B 0,C 180,E1 19528.014,E2 19528.014} C_VEL
LIN {X 0,Y 391.944,Z 1176.802,A -85,B 0,C 180,E1 19527.606,E2 19527.606} C_VEL
LIN {X 0,Y 392.014,Z 1175.231,A -85,B 0,C 180,E1 19523.85,E2 19523.85} C_VEL
LIN {X 0,Y 392.229,Z 1172.349,A -85,B 0,C 180,E1 19520.314,E2 19520.314} C_VEL
LIN {X 0,Y 392.709,Z 1168.601,A -85,B 0,C 180,E1 19517.053,E2 19517.053} C_VEL
LIN {X 0,Y 393.573,Z 1163.98,A -85,B 0,C 180,E1 19513.924,E2 19513.924} C_VEL
LIN {X 0,Y 394.919,Z 1158.298,A -85,B 0,C 180,E1 19510.784,E2 19510.784} C_VEL
LIN {X 0,Y 396.995,Z 1151.165,A -85,B 0,C 180,E1 19507.492,E2 19507.492} C_VEL
LIN {X 0,Y 400.557,Z 1140.646,A -85,B 0,C 180,E1 19503.461,E2 19503.461} C_VEL
LIN {X 0,Y 404.606,Z 1129.928,A -85,B 0,C 180,E1 19500.054,E2 19500.054} C_VEL
LIN {X 0,Y 408.683,Z 1119.866,A -85,B 0,C 180,E1 19497.27,E2 19497.27} C_VEL
LIN {X 0,Y 413.498,Z 1108.578,A -85,B 0,C 180,E1 19494.526,E2 19494.526} C_VEL
LIN {X 0,Y 420.013,Z 1093.888,A -85,B 0,C 180,E1 19491.413,E2 19491.413} C_VEL
LIN {X 0,Y 427.437,Z 1076.953,A -85,B 0,C 180,E1 19488.369,E2 19488.369} C_VEL
LIN {X 0,Y 434.055,Z 1061.833,A -85,B 0,C 180,E1 19486.012,E2 19486.012} C_VEL
LIN {X 0,Y 440.606,Z 1046.612,A -85,B 0,C 180,E1 19483.923,E2 19483.923} C_VEL
LIN {X 0,Y 447.978,Z 1028.997,A -85,B 0,C 180,E1 19481.801,E2 19481.801} C_VEL
LIN {X 0,Y 457.028,Z 1006.049,A -85,B 0,C 180,E1 19479.442,E2 19479.442} C_VEL
LIN {X 0,Y 463.88,Z 987.563,A -85,B 0,C 180,E1 19477.818,E2 19477.818} C_VEL
LIN {X 0,Y 469.979,Z 970.054,A -85,B 0,C 180,E1 19476.469,E2 19476.469} C_VEL
LIN {X 0,Y 475.995,Z 951.382,A -85,B 0,C 180,E1 19475.203,E2 19475.203} C_VEL
LIN {X 0,Y 482.221,Z 930.324,A -85,B 0,C 180,E1 19473.966,E2 19473.966} C_VEL
LIN {X 0,Y 489.239,Z 903.413,A -85,B 0,C 180,E1 19472.648,E2 19472.648} C_VEL
LIN {X 0,Y 494.192,Z 881.266,A -85,B 0,C 180,E1 19471.757,E2 19471.757} C_VEL
LIN {X 0,Y 498.255,Z 860.18,A -85,B 0,C 180,E1 19471.049,E2 19471.049} C_VEL
LIN {X 0,Y 501.736,Z 838.658,A -85,B 0,C 180,E1 19470.457,E2 19470.457} C_VEL
LIN {X 0,Y 505.082,Z 812.635,A -85,B 0,C 180,E1 19469.897,E2 19469.897} C_VEL
LIN {X 0,Y 508.083,Z 772.485,A -85,B 0,C 180,E1 19469.244,E2 19469.244} C_VEL
LIN {X 0,Y 522.75,Z 550.207,A -85,B 0,C 180,E1 19465.787,E2 19465.787} C_VEL
LIN {X 0,Y 525.891,Z 503.895,A -85,B 0,C 180,E1 19465.057,E2 19465.057} C_VEL
LIN {X 0,Y 517.841,Z 491.671,A -85,B 0,C 180,E1 19462.627,E2 19462.627} C_VEL
LIN {X 0,Y 509.965,Z 480.396,A -85,B 0,C 180,E1 19459.918,E2 19459.918} C_VEL
LIN {X 0,Y 504.024,Z 472.048,A -85,B 0,C 180,E1 19457.55,E2 19457.55} C_VEL
LIN {X 0,Y 500.103,Z 466.848,A -85,B 0,C 180,E1 19455.778,E2 19455.778} C_VEL
LIN {X 0,Y 496.383,Z 461.892,A -85,B 0,C 180,E1 19453.86,E2 19453.86} C_VEL
LIN {X 0,Y 493.029,Z 457.169,A -85,B 0,C 180,E1 19451.82,E2 19451.82} C_VEL
LIN {X 0,Y 489.498,Z 453.032,A -85,B 0,C 180,E1 19449.227,E2 19449.227} C_VEL
LIN {X 0,Y 488.467,Z 451.153,A -85,B 0,C 180,E1 19448.238,E2 19448.238} C_VEL
LIN {X 0,Y 485.308,Z 447.716,A -85,B 0,C 180,E1 19444.254,E2 19444.254} C_VEL
LIN {X 0,Y 484.704,Z 445.286,A -85,B 0,C 180,E1 19442.246,E2 19442.246} C_VEL
LIN {X 0,Y 484.771,Z 445.528,A -85,B 0,C 180,E1 19437.872,E2 19437.872} C_VEL
LIN {X 0,Y 486.708,Z 449.824,A -85,B 0,C 180,E1 19433.986,E2 19433.986} C_VEL
LIN {X 0,Y 488.909,Z 451.665,A -85,B 0,C 180,E1 19431.769,E2 19431.769} C_VEL
LIN {X 0,Y 491.718,Z 455.998,A -85,B 0,C 180,E1 19429.455,E2 19429.455} C_VEL
LIN {X 0,Y 493.368,Z 457.754,A -85,B 0,C 180,E1 19428.366,E2 19428.366} C_VEL
LIN {X 0,Y 497.557,Z 463.356,A -85,B 0,C 180,E1 19425.927,E2 19425.927} C_VEL
LIN {X 0,Y 502.13,Z 469.597,A -85,B 0,C 180,E1 19423.693,E2 19423.693} C_VEL
LIN {X 0,Y 508.144,Z 478.903,A -85,B 0,C 180,E1 19421.143,E2 19421.143} C_VEL
LIN {X 0,Y 514.427,Z 488.859,A -85,B 0,C 180,E1 19418.836,E2 19418.836} C_VEL
LIN {X 0,Y 522.369,Z 502.051,A -85,B 0,C 180,E1 19416.268,E2 19416.268} C_VEL
LIN {X 0,Y 525.976,Z 508.458,A -85,B 0,C 180,E1 19415.195,E2 19415.195} C_VEL
LIN {X 0,Y 511.366,Z 728.014,A -85,B 0,C 180,E1 19411.777,E2 19411.777} C_VEL
LIN {X 0,Y 505.204,Z 821.158,A -85,B 0,C 180,E1 19410.309,E2 19410.309} C_VEL
LIN {X 0,Y 502.051,Z 849.003,A -85,B 0,C 180,E1 19409.778,E2 19409.778} C_VEL
LIN {X 0,Y 497.809,Z 874.979,A -85,B 0,C 180,E1 19409.122,E2 19409.122} C_VEL
LIN {X 0,Y 493.674,Z 896.256,A -85,B 0,C 180,E1 19408.447,E2 19408.447} C_VEL
LIN {X 0,Y 489.189,Z 916.28,A -85,B 0,C 180,E1 19407.688,E2 19407.688} C_VEL
LIN {X 0,Y 484.064,Z 936.652,A -85,B 0,C 180,E1 19406.777,E2 19406.777} C_VEL
LIN {X 0,Y 477.075,Z 961.674,A -85,B 0,C 180,E1 19405.452,E2 19405.452} C_VEL
LIN {X 0,Y 469.475,Z 985.513,A -85,B 0,C 180,E1 19403.924,E2 19403.924} C_VEL
LIN {X 0,Y 462.776,Z 1005.097,A -85,B 0,C 180,E1 19402.46,E2 19402.46} C_VEL
LIN {X 0,Y 456.13,Z 1023.388,A -85,B 0,C 180,E1 19400.894,E2 19400.894} C_VEL
LIN {X 0,Y 448.396,Z 1043.627,A -85,B 0,C 180,E1 19398.911,E2 19398.911} C_VEL
LIN {X 0,Y 439.752,Z 1064.954,A -85,B 0,C 180,E1 19396.453,E2 19396.453} C_VEL
LIN {X 0,Y 432.835,Z 1081.577,A -85,B 0,C 180,E1 19394.237,E2 19394.237} C_VEL
LIN {X 0,Y 426.432,Z 1096.799,A -85,B 0,C 180,E1 19391.931,E2 19391.931} C_VEL
LIN {X 0,Y 419.279,Z 1113.912,A -85,B 0,C 180,E1 19388.973,E2 19388.973} C_VEL
LIN {X 0,Y 412.664,Z 1129.827,A -85,B 0,C 180,E1 19385.727,E2 19385.727} C_VEL
LIN {X 0,Y 407.684,Z 1142.244,A -85,B 0,C 180,E1 19382.82,E2 19382.82} C_VEL
LIN {X 0,Y 403.717,Z 1152.77,A -85,B 0,C 180,E1 19380.018,E2 19380.018} C_VEL
LIN {X 0,Y 400.093,Z 1163.207,A -85,B 0,C 180,E1 19376.849,E2 19376.849} C_VEL
LIN {X 0,Y 396.517,Z 1174.883,A -85,B 0,C 180,E1 19372.64,E2 19372.64} C_VEL
LIN {X 0,Y 394.595,Z 1182.366,A -85,B 0,C 180,E1 19369.386,E2 19369.386} C_VEL
LIN {X 0,Y 393.333,Z 1188.461,A -85,B 0,C 180,E1 19366.238,E2 19366.238} C_VEL
LIN {X 0,Y 392.573,Z 1193.232,A -85,B 0,C 180,E1 19363.251,E2 19363.251} C_VEL
LIN {X 0,Y 392.165,Z 1197.102,A -85,B 0,C 180,E1 19360.206,E2 19360.206} C_VEL
LIN {X 0,Y 392.003,Z 1199.843,A -85,B 0,C 180,E1 19357.327,E2 19357.327} C_VEL
LIN {X 0,Y 391.941,Z 1201.717,A -85,B 0,C 180,E1 19354.389,E2 19354.389} C_VEL
LIN {X 0,Y 391.942,Z 1202.63,A -85,B 0,C 180,E1 19351.608,E2 19351.608} C_VEL
LIN {X 0,Y 391.944,Z 1202.7,A -85,B 0,C 180,E1 19348.831,E2 19348.831} C_VEL
LIN {X 0,Y 391.94,Z 1201.857,A -85,B 0,C 180,E1 19345.904,E2 19345.904} C_VEL
LIN {X 0,Y 391.984,Z 1200.076,A -85,B 0,C 180,E1 19342.967,E2 19342.967} C_VEL
LIN {X 0,Y 392.147,Z 1197.347,A -85,B 0,C 180,E1 19340.016,E2 19340.016} C_VEL
LIN {X 0,Y 392.516,Z 1193.656,A -85,B 0,C 180,E1 19337.046,E2 19337.046} C_VEL
LIN {X 0,Y 393.277,Z 1188.799,A -85,B 0,C 180,E1 19333.957,E2 19333.957} C_VEL
LIN {X 0,Y 394.443,Z 1182.985,A -85,B 0,C 180,E1 19330.913,E2 19330.913} C_VEL
LIN {X 0,Y 396.246,Z 1175.84,A -85,B 0,C 180,E1 19327.759,E2 19327.759} C_VEL
LIN {X 0,Y 399.263,Z 1165.838,A -85,B 0,C 180,E1 19324.008,E2 19324.008} C_VEL
LIN {X 0,Y 403.351,Z 1153.817,A -85,B 0,C 180,E1 19320.279,E2 19320.279} C_VEL
LIN {X 0,Y 407.462,Z 1142.799,A -85,B 0,C 180,E1 19317.321,E2 19317.321} C_VEL
LIN {X 0,Y 412.116,Z 1131.103,A -85,B 0,C 180,E1 19314.56,E2 19314.56} C_VEL
LIN {X 0,Y 417.817,Z 1117.323,A -85,B 0,C 180,E1 19311.699,E2 19311.699} C_VEL
LIN {X 0,Y 425.713,Z 1098.476,A -85,B 0,C 180,E1 19308.343,E2 19308.343} C_VEL
LIN {X 0,Y 432.431,Z 1082.468,A -85,B 0,C 180,E1 19305.896,E2 19305.896} C_VEL
LIN {X 0,Y 438.973,Z 1066.726,A -85,B 0,C 180,E1 19303.777,E2 19303.777} C_VEL
LIN {X 0,Y 446.51,Z 1048.2,A -85,B 0,C 180,E1 19301.59,E2 19301.59} C_VEL
LIN {X 0,Y 455.366,Z 1025.313,A -85,B 0,C 180,E1 19299.286,E2 19299.286} C_VEL
LIN {X 0,Y 462.235,Z 1006.463,A -85,B 0,C 180,E1 19297.656,E2 19297.656} C_VEL
LIN {X 0,Y 468.79,Z 987.386,A -85,B 0,C 180,E1 19296.215,E2 19296.215} C_VEL
LIN {X 0,Y 475.341,Z 966.987,A -85,B 0,C 180,E1 19294.881,E2 19294.881} C_VEL
LIN {X 0,Y 482.584,Z 942.153,A -85,B 0,C 180,E1 19293.495,E2 19293.495} C_VEL
LIN {X 0,Y 488.646,Z 918.282,A -85,B 0,C 180,E1 19292.4,E2 19292.4} C_VEL
LIN {X 0,Y 493.345,Z 897.475,A -85,B 0,C 180,E1 19291.601,E2 19291.601} C_VEL
LIN {X 0,Y 497.55,Z 875.967,A -85,B 0,C 180,E1 19290.912,E2 19290.912} C_VEL
LIN {X 0,Y 501.355,Z 852.924,A -85,B 0,C 180,E1 19290.32,E2 19290.32} C_VEL
LIN {X 0,Y 504.997,Z 822.639,A -85,B 0,C 180,E1 19289.722,E2 19289.722} C_VEL
LIN {X 0,Y 509.347,Z 758.142,A -85,B 0,C 180,E1 19288.698,E2 19288.698} C_VEL
LIN {X 0,Y 523.92,Z 537.057,A -85,B 0,C 180,E1 19285.258,E2 19285.258} C_VEL
LIN {X 0,Y 525.824,Z 508.148,A -85,B 0,C 180,E1 19284.79,E2 19284.79} C_VEL
LIN {X 0,Y 518.336,Z 495.451,A -85,B 0,C 180,E1 19282.514,E2 19282.514} C_VEL
LIN {X 0,Y 511.078,Z 483.542,A -85,B 0,C 180,E1 19280.022,E2 19280.022} C_VEL
LIN {X 0,Y 504.46,Z 473.349,A -85,B 0,C 180,E1 19277.415,E2 19277.415} C_VEL
LIN {X 0,Y 500.422,Z 467.247,A -85,B 0,C 180,E1 19275.59,E2 19275.59} C_VEL
LIN {X 0,Y 496.235,Z 461.699,A -85,B 0,C 180,E1 19273.458,E2 19273.458} C_VEL
LIN {X 0,Y 492.571,Z 456.779,A -85,B 0,C 180,E1 19271.237,E2 19271.237} C_VEL
LIN {X 0,Y 489.512,Z 453.058,A -85,B 0,C 180,E1 19268.99,E2 19268.99} C_VEL
LIN {X 0,Y 488.583,Z 451.247,A -85,B 0,C 180,E1 19268.118,E2 19268.118} C_VEL
LIN {X 0,Y 485.364,Z 447.937,A -85,B 0,C 180,E1 19264.372,E2 19264.372} C_VEL
LIN {X 0,Y 484.531,Z 445.262,A -85,B 0,C 180,E1 19262.129,E2 19262.129} C_VEL
LIN {X 0,Y 484.636,Z 445.392,A -85,B 0,C 180,E1 19257.043,E2 19257.043} C_VEL
LIN {X 0,Y 485.852,Z 448.759,A -85,B 0,C 180,E1 19254.331,E2 19254.331} C_VEL
LIN {X 0,Y 488.727,Z 451.543,A -85,B 0,C 180,E1 19251.233,E2 19251.233} C_VEL
LIN {X 0,Y 491.318,Z 455.593,A -85,B 0,C 180,E1 19249.09,E2 19249.09} C_VEL
LIN {X 0,Y 493.137,Z 457.512,A -85,B 0,C 180,E1 19247.886,E2 19247.886} C_VEL
LIN {X 0,Y 496.49,Z 462.026,A -85,B 0,C 180,E1 19245.896,E2 19245.896} C_VEL
LIN {X 0,Y 501.555,Z 468.791,A -85,B 0,C 180,E1 19243.377,E2 19243.377} C_VEL
LIN {X 0,Y 505.905,Z 474.833,A -85,B 0,C 180,E1 19241.505,E2 19241.505} C_VEL
LIN {X 0,Y 511.612,Z 482.702,A -85,B 0,C 180,E1 19239.343,E2 19239.343} C_VEL
LIN {X 0,Y 520.881,Z 496.234,A -85,B 0,C 180,E1 19236.294,E2 19236.294} C_VEL
LIN {X 0,Y 525.804,Z 504.161,A -85,B 0,C 180,E1 19234.834,E2 19234.834} C_VEL
LIN {X 0,Y 511.352,Z 720.193,A -85,B 0,C 180,E1 19231.475,E2 19231.475} C_VEL
LIN {X 0,Y 505.677,Z 804.917,A -85,B 0,C 180,E1 19230.14,E2 19230.14} C_VEL
LIN {X 0,Y 502.556,Z 832.706,A -85,B 0,C 180,E1 19229.595,E2 19229.595} C_VEL
LIN {X 0,Y 498.567,Z 858.001,A -85,B 0,C 180,E1 19228.921,E2 19228.921} C_VEL
LIN {X 0,Y 494.554,Z 879.104,A -85,B 0,C 180,E1 19228.227,E2 19228.227} C_VEL
LIN {X 0,Y 490.055,Z 899.569,A -85,B 0,C 180,E1 19227.42,E2 19227.42} C_VEL
LIN {X 0,Y 484.471,Z 921.877,A -85,B 0,C 180,E1 19226.382,E2 19226.382} C_VEL
LIN {X 0,Y 477.102,Z 947.696,A -85,B 0,C 180,E1 19224.932,E2 19224.932} C_VEL
LIN {X 0,Y 470.737,Z 967.604,A -85,B 0,C 180,E1 19223.611,E2 19223.611} C_VEL
LIN {X 0,Y 464.35,Z 986.063,A -85,B 0,C 180,E1 19222.208,E2 19222.208} C_VEL
LIN {X 0,Y 457.725,Z 1004.02,A -85,B 0,C 180,E1 19220.649,E2 19220.649} C_VEL
LIN {X 0,Y 450.026,Z 1023.841,A -85,B 0,C 180,E1 19218.673,E2 19218.673} C_VEL
LIN {X 0,Y 441.267,Z 1044.973,A -85,B 0,C 180,E1 19216.193,E2 19216.193} C_VEL
LIN {X 0,Y 434.433,Z 1060.876,A -85,B 0,C 180,E1 19214.032,E2 19214.032} C_VEL
LIN {X 0,Y 427.966,Z 1075.658,A -85,B 0,C 180,E1 19211.747,E2 19211.747} C_VEL
LIN {X 0,Y 421.123,Z 1091.276,A -85,B 0,C 180,E1 19208.99,E2 19208.99} C_VEL
LIN {X 0,Y 413.925,Z 1107.601,A -85,B 0,C 180,E1 19205.602,E2 19205.602} C_VEL
LIN {X 0,Y 409.043,Z 1118.986,A -85,B 0,C 180,E1 19202.864,E2 19202.864} C_VEL
LIN {X 0,Y 404.911,Z 1129.137,A -85,B 0,C 180,E1 19200.084,E2 19200.084} C_VEL
LIN {X 0,Y 401.278,Z 1138.592,A -85,B 0,C 180,E1 19197.128,E2 19197.128} C_VEL
LIN {X 0,Y 397.781,Z 1148.751,A -85,B 0,C 180,E1 19193.438,E2 19193.438} C_VEL
LIN {X 0,Y 395.128,Z 1157.529,A -85,B 0,C 180,E1 19189.513,E2 19189.513} C_VEL
LIN {X 0,Y 393.66,Z 1163.583,A -85,B 0,C 180,E1 19186.224,E2 19186.224} C_VEL
LIN {X 0,Y 392.753,Z 1168.278,A -85,B 0,C 180,E1 19183.095,E2 19183.095} C_VEL
LIN {X 0,Y 392.269,Z 1171.943,A -85,B 0,C 180,E1 19179.981,E2 19179.981} C_VEL
LIN {X 0,Y 392.041,Z 1174.611,A -85,B 0,C 180,E1 19176.884,E2 19176.884} C_VEL
LIN {X 0,Y 391.958,Z 1176.37,A -85,B 0,C 180,E1 19173.656,E2 19173.656} C_VEL
LIN {X 0,Y 391.939,Z 1177.14,A -85,B 0,C 180,E1 19169.854,E2 19169.854} C_VEL
LIN {X 0,Y 391.944,Z 1176.802,A -85,B 0,C 180,E1 19167.606,E2 19167.606} C_VEL
LIN {X 0,Y 390.958,Z 1176.573,A -85,B 0,C 180,E1 19166.48,E2 19166.48} C_VEL
LIN {X 0,Y 384.586,Z 1175.182,A -85,B 0,C 180,E1 19163.309,E2 19163.309} C_VEL
LIN {X 0,Y 384.075,Z 1174.587,A -85,B 0,C 180,E1 19162.483,E2 19162.483} C_VEL
LIN {X 0,Y 384.328,Z 1171.996,A -85,B 0,C 180,E1 19159.507,E2 19159.507} C_VEL
LIN {X 0,Y 384.893,Z 1168.267,A -85,B 0,C 180,E1 19156.326,E2 19156.326} C_VEL
LIN {X 0,Y 385.876,Z 1163.509,A -85,B 0,C 180,E1 19153.13,E2 19153.13} C_VEL
LIN {X 0,Y 387.716,Z 1156.704,A -85,B 0,C 180,E1 19149.416,E2 19149.416} C_VEL
LIN {X 0,Y 390.745,Z 1147.38,A -85,B 0,C 180,E1 19145.349,E2 19145.349} C_VEL
LIN {X 0,Y 393.973,Z 1138.677,A -85,B 0,C 180,E1 19142.162,E2 19142.162} C_VEL
LIN {X 0,Y 397.803,Z 1129.194,A -85,B 0,C 180,E1 19139.153,E2 19139.153} C_VEL
LIN {X 0,Y 402.732,Z 1117.83,A -85,B 0,C 180,E1 19136.022,E2 19136.022} C_VEL
LIN {X 0,Y 409.982,Z 1101.726,A -85,B 0,C 180,E1 19132.256,E2 19132.256} C_VEL
LIN {X 0,Y 416.192,Z 1088.188,A -85,B 0,C 180,E1 19129.561,E2 19129.561} C_VEL
LIN {X 0,Y 422.373,Z 1074.728,A -85,B 0,C 180,E1 19127.204,E2 19127.204} C_VEL
LIN {X 0,Y 429.136,Z 1059.822,A -85,B 0,C 180,E1 19124.904,E2 19124.904} C_VEL
LIN {X 0,Y 437.875,Z 1040.224,A -85,B 0,C 180,E1 19122.283,E2 19122.283} C_VEL
LIN {X 0,Y 445.872,Z 1021.148,A -85,B 0,C 180,E1 19120.121,E2 19120.121} C_VEL
LIN {X 0,Y 452.866,Z 1003.672,A -85,B 0,C 180,E1 19118.392,E2 19118.392} C_VEL
LIN {X 0,Y 459.696,Z 985.645,A -85,B 0,C 180,E1 19116.83,E2 19116.83} C_VEL
LIN {X 0,Y 466.667,Z 965.967,A -85,B 0,C 180,E1 19115.346,E2 19115.346} C_VEL
LIN {X 0,Y 474.826,Z 940.557,A -85,B 0,C 180,E1 19113.72,E2 19113.72} C_VEL
LIN {X 0,Y 480.968,Z 918.895,A -85,B 0,C 180,E1 19112.556,E2 19112.556} C_VEL
LIN {X 0,Y 486.145,Z 898.561,A -85,B 0,C 180,E1 19111.628,E2 19111.628} C_VEL
LIN {X 0,Y 490.762,Z 877.89,A -85,B 0,C 180,E1 19110.824,E2 19110.824} C_VEL
LIN {X 0,Y 495.586,Z 852.71,A -85,B 0,C 180,E1 19110.02,E2 19110.02} C_VEL
LIN {X 0,Y 499.586,Z 825.475,A -85,B 0,C 180,E1 19109.355,E2 19109.355} C_VEL
LIN {X 0,Y 502.052,Z 802.61,A -85,B 0,C 180,E1 19108.928,E2 19108.928} C_VEL
LIN {X 0,Y 516.426,Z 591.9,A -85,B 0,C 180,E1 19105.636,E2 19105.636} C_VEL
LIN {X 0,Y 522.226,Z 508.876,A -85,B 0,C 180,E1 19104.339,E2 19104.339} C_VEL
LIN {X 0,Y 515.379,Z 498.381,A -85,B 0,C 180,E1 19102.2,E2 19102.2} C_VEL
LIN {X 0,Y 507.967,Z 487.556,A -85,B 0,C 180,E1 19099.58,E2 19099.58} C_VEL
LIN {X 0,Y 502.143,Z 479.285,A -85,B 0,C 180,E1 19097.2,E2 19097.2} C_VEL
LIN {X 0,Y 498.543,Z 474.405,A -85,B 0,C 180,E1 19095.531,E2 19095.531} C_VEL
LIN {X 0,Y 494.909,Z 469.499,A -85,B 0,C 180,E1 19093.614,E2 19093.614} C_VEL
LIN {X 0,Y 491.353,Z 464.532,A -85,B 0,C 180,E1 19091.385,E2 19091.385} C_VEL
LIN {X 0,Y 488.256,Z 460.722,A -85,B 0,C 180,E1 19089.013,E2 19089.013} C_VEL
LIN {X 0,Y 487.369,Z 459.041,A -85,B 0,C 180,E1 19088.138,E2 19088.138} C_VEL
LIN {X 0,Y 484.223,Z 455.46,A -85,B 0,C 180,E1 19084.026,E2 19084.026} C_VEL
LIN {X 0,Y 483.696,Z 453.224,A -85,B 0,C 180,E1 19082.132,E2 19082.132} C_VEL
LIN {X 0,Y 483.763,Z 453.413,A -85,B 0,C 180,E1 19077.986,E2 19077.986} C_VEL
LIN {X 0,Y 485.638,Z 457.706,A -85,B 0,C 180,E1 19074.091,E2 19074.091} C_VEL
LIN {X 0,Y 487.796,Z 459.616,A -85,B 0,C 180,E1 19071.869,E2 19071.869} C_VEL
LIN {X 0,Y 490.581,Z 463.882,A -85,B 0,C 180,E1 19069.549,E2 19069.549} C_VEL
LIN {X 0,Y 492.035,Z 465.449,A -85,B 0,C 180,E1 19068.572,E2 19068.572} C_VEL
LIN {X 0,Y 496.148,Z 471.071,A -85,B 0,C 180,E1 19066.124,E2 19066.124} C_VEL
LIN {X 0,Y 500.534,Z 477.139,A -85,B 0,C 180,E1 19063.938,E2 19063.938} C_VEL
LIN {X 0,Y 507.147,Z 487.482,A -85,B 0,C 180,E1 19061.105,E2 19061.105} C_VEL
